FUNCTION_BLOCK "HF3_3#SB_FB2562"	// FB 2562
VERSION : 0.1
VAR_INPUT
  SCtrl : WORD ;	//上位控制命令
  inRD : ARRAY  [0 .. 3 ] OF //输入状态字
  WORD ;
  PT24 : TIME ;	//超时时间
  H_P_ALL_Ctrl : WORD ;	//全局控制命令
END_VAR
VAR_OUTPUT
  qnWR : WORD ;	//控制命令
  ToHMI1 : WORD ;	//反馈上位信息1
  ToHMI2 : WORD ;	//反馈上位信息2
  RT1 : INT ;	//1泵运行时间
  RT2 : INT ;	//2泵运行时间
  RT3 : INT ;
  SumFlt1 : INT ;	//1泵故障次数
  SumFlt2 : INT ;	//2泵故障次数
  SumFlt3 : INT ;
  SumRun1 : INT ;	//1泵运行次数
  SumRun2 : INT ;	//2泵运行次数
  SumRun3 : INT ;
  Level_Value : INT ;	//水位mm
END_VAR
VAR
  Ton1 : SFB 4;
  Ton2 : SFB 4;
  Ton3 : SFB 4;
  Ton4 : SFB 4;
  Ton5 : SFB 4;
  Ton6 : SFB 4;
  Ton7 : SFB 4;
  SingTout1 : BOOL ;	//一泵控制超时
  SingTout2 : BOOL ;	//二泵控制超时
  SingTout3 : BOOL ;	//三泵控制超时
  Timeout1 : BOOL ;	//一泵超时
  Timeout2 : BOOL ;	//二泵超时
  Timeout3 : BOOL ;	//三泵超时
  DI_Temp1 : ARRAY  [0 .. 15 ] OF //0自动1-1运行5-2运行9-3运行
  BOOL ;
  DI_Temp2 : ARRAY  [0 .. 15 ] OF //水泵状态字
  BOOL ;
  DO_Temp : ARRAY  [0 .. 15 ] OF //01-1泵启停23-2泵启停45-3泵启停
  BOOL ;
  Ctrl : ARRAY  [0 .. 15 ] OF //01-1泵启停23-2泵启停45-3泵启停
  BOOL ;
  SCtrl_Temp : ARRAY  [0 .. 15 ] OF //01-1泵启停23-2泵启停45-3泵启停6-3泵同启
  BOOL ;
  Latch : ARRAY  [0 .. 7 ] OF //01-1泵启停锁定23-2泵启停锁定45-3泵启停锁定
  BOOL ;
  McFlag : BOOL ;	//挂检修牌
  QTout1 : BOOL ;	//一泵输出超时
  QTout2 : BOOL ;	//二泵输出超时
  QTout3 : BOOL ;	//三泵输出超时
  H_P_ALL_Ctrl_Temp : ARRAY  [0 .. 15 ] OF BOOL ;
  CommOK_Temp : ARRAY  [0 .. 15 ] OF //通信中间变量
  BOOL ;
  CommOK : BOOL ;	//通信正常
END_VAR
BEGIN
NETWORK
TITLE =
      A(;
      BLD   1;
      =     L 4.0;
      TAR2  LD 0;
      L     #SCtrl;
      T     LW 5;
      L     DINO;
      T     LW 7;
      +AR2  P#206.0;
      TAR2;
      LAR2  LD 0;
      T     LD 9;
      UC    "HF3_W_T_B_FC54";
      {     P#L 5.0, P#L 7.0 };
      LAR2  LD 0;
      BLD   2;
      A     BR;
      );
      JNB   _001;
      BLD   1;
      =     L 4.0;
      TAR2  LD 0;
      L     #H_P_ALL_Ctrl;
      T     LW 5;
      L     DINO;
      T     LW 7;
      +AR2  P#212.0;
      TAR2;
      LAR2  LD 0;
      T     LD 9;
      UC    "HF3_W_T_B_FC54";
      {     P#L 5.0, P#L 7.0 };
      LAR2  LD 0;
      BLD   2;
_001: NOP   0;
NETWORK
TITLE =
      A(;
      BLD   1;
      =     L 4.0;
      TAR2  LD 0;
      L     #inRD[1];
      T     LW 5;
      L     DINO;
      T     LW 7;
      +AR2  P#198.0;
      TAR2;
      LAR2  LD 0;
      T     LD 9;
      UC    "HF3_W_T_B_FC54";
      {     P#L 5.0, P#L 7.0 };
      LAR2  LD 0;
      BLD   2;
      A     BR;
      );
      JNB   _002;
      BLD   1;
      =     L 4.0;
      TAR2  LD 0;
      L     #inRD[2];
      T     LW 5;
      L     DINO;
      T     LW 7;
      +AR2  P#200.0;
      TAR2;
      LAR2  LD 0;
      T     LD 9;
      UC    "HF3_W_T_B_FC54";
      {     P#L 5.0, P#L 7.0 };
      LAR2  LD 0;
      BLD   2;
_002: NOP   0;
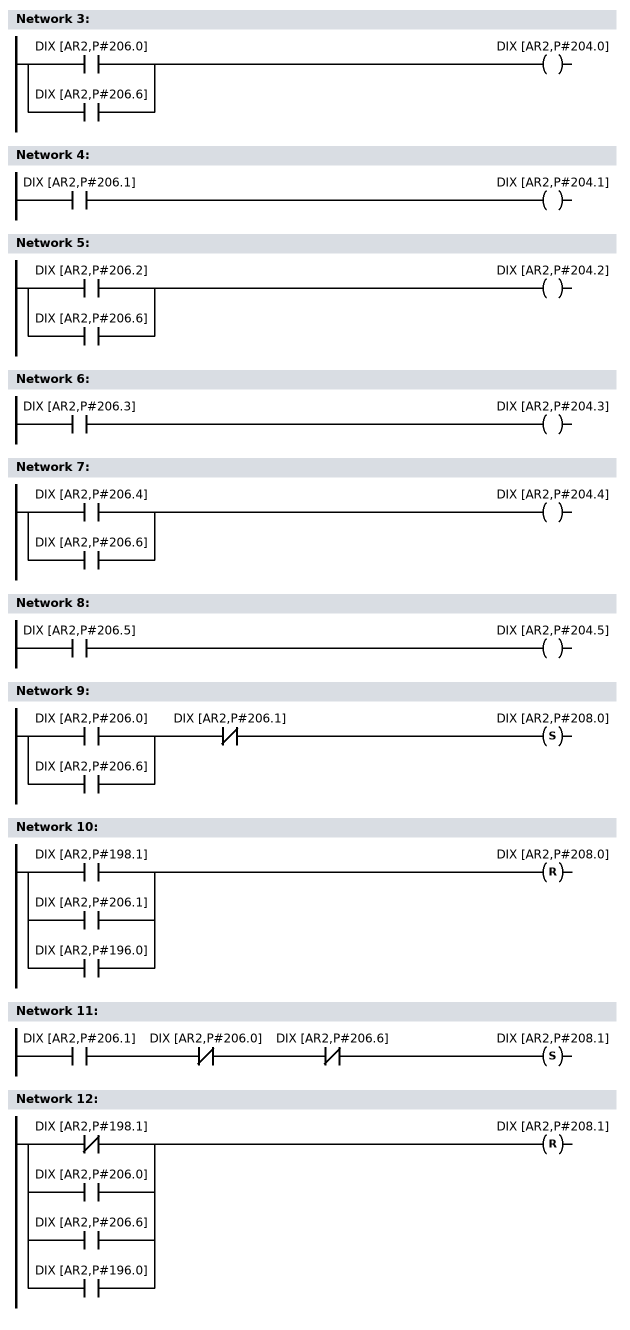
NETWORK
TITLE =
      O     DIX [AR2,P#206.0];
      O     DIX [AR2,P#206.6];
      =     DIX [AR2,P#204.0];
NETWORK
TITLE =
      A     DIX [AR2,P#206.1];
      =     DIX [AR2,P#204.1];
NETWORK
TITLE =
      O     DIX [AR2,P#206.2];
      O     DIX [AR2,P#206.6];
      =     DIX [AR2,P#204.2];
NETWORK
TITLE =
      A     DIX [AR2,P#206.3];
      =     DIX [AR2,P#204.3];
NETWORK
TITLE =
      O     DIX [AR2,P#206.4];
      O     DIX [AR2,P#206.6];
      =     DIX [AR2,P#204.4];
NETWORK
TITLE =
      A     DIX [AR2,P#206.5];
      =     DIX [AR2,P#204.5];
NETWORK
TITLE =
      A(;
      O     DIX [AR2,P#206.0];
      O     DIX [AR2,P#206.6];
      );
      AN    DIX [AR2,P#206.1];
      S     DIX [AR2,P#208.0];
NETWORK
TITLE =
      O     DIX [AR2,P#198.1];
      O     DIX [AR2,P#206.1];
      O     DIX [AR2,P#196.0];
      R     DIX [AR2,P#208.0];
NETWORK
TITLE =
      A     DIX [AR2,P#206.1];
      AN    DIX [AR2,P#206.0];
      AN    DIX [AR2,P#206.6];
      S     DIX [AR2,P#208.1];
NETWORK
TITLE =
      ON    DIX [AR2,P#198.1];
      O     DIX [AR2,P#206.0];
      O     DIX [AR2,P#206.6];
      O     DIX [AR2,P#196.0];
      R     DIX [AR2,P#208.1];
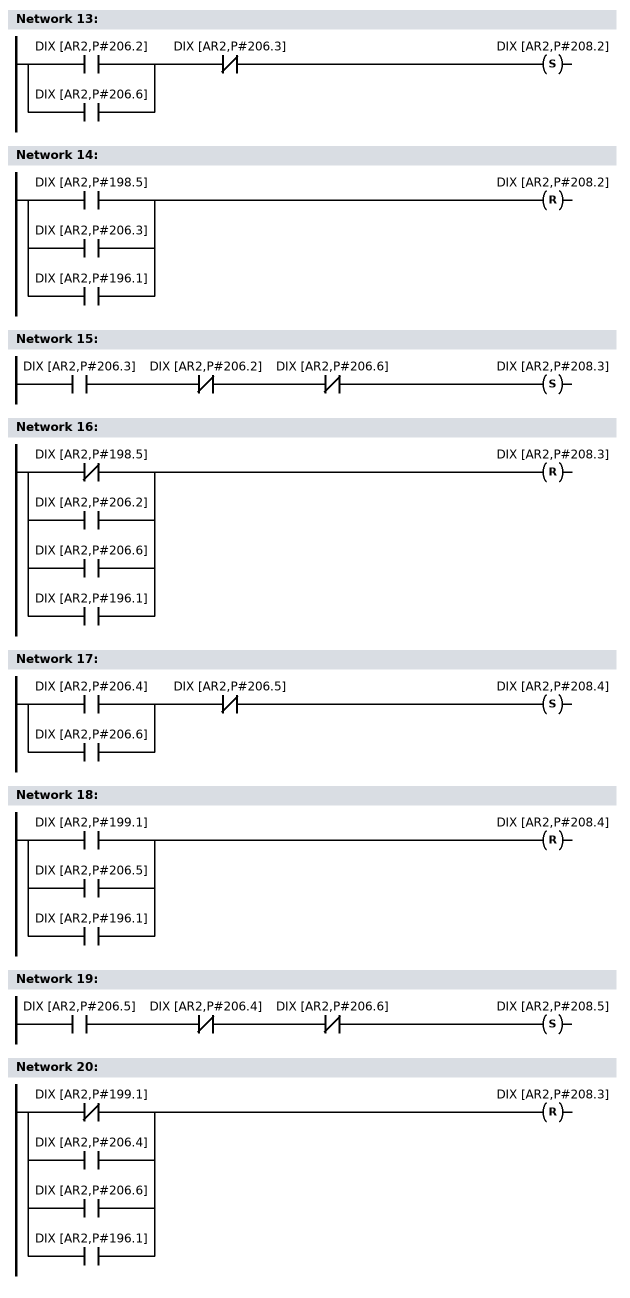
NETWORK
TITLE =
      A(;
      O     DIX [AR2,P#206.2];
      O     DIX [AR2,P#206.6];
      );
      AN    DIX [AR2,P#206.3];
      S     DIX [AR2,P#208.2];
NETWORK
TITLE =
      O     DIX [AR2,P#198.5];
      O     DIX [AR2,P#206.3];
      O     DIX [AR2,P#196.1];
      R     DIX [AR2,P#208.2];
NETWORK
TITLE =
      A     DIX [AR2,P#206.3];
      AN    DIX [AR2,P#206.2];
      AN    DIX [AR2,P#206.6];
      S     DIX [AR2,P#208.3];
NETWORK
TITLE =
      ON    DIX [AR2,P#198.5];
      O     DIX [AR2,P#206.2];
      O     DIX [AR2,P#206.6];
      O     DIX [AR2,P#196.1];
      R     DIX [AR2,P#208.3];
NETWORK
TITLE =
      A(;
      O     DIX [AR2,P#206.4];
      O     DIX [AR2,P#206.6];
      );
      AN    DIX [AR2,P#206.5];
      S     DIX [AR2,P#208.4];
NETWORK
TITLE =
      O     DIX [AR2,P#199.1];
      O     DIX [AR2,P#206.5];
      O     DIX [AR2,P#196.1];
      R     DIX [AR2,P#208.4];
NETWORK
TITLE =
      A     DIX [AR2,P#206.5];
      AN    DIX [AR2,P#206.4];
      AN    DIX [AR2,P#206.6];
      S     DIX [AR2,P#208.5];
NETWORK
TITLE =
      ON    DIX [AR2,P#199.1];
      O     DIX [AR2,P#206.4];
      O     DIX [AR2,P#206.6];
      O     DIX [AR2,P#196.1];
      R     DIX [AR2,P#208.3];
NETWORK
TITLE =
      A(;
      O     DIX [AR2,P#208.0];
      O     DIX [AR2,P#208.1];
      );
      AN    DIX [AR2,P#206.0];
      AN    DIX [AR2,P#206.1];
      AN    DIX [AR2,P#206.6];
      =     L 0.0;
      BLD   103;
      BLD   16;
      =     L 7.0;
      L     DINO;
      T     LW 5;
      CDB;
      OPN   DI [LW 5];
      TAR2  LD 1;
      A     L 0.0;
      =     DIX [AR2,P#42.0];
      L     DBD [AR2,P#10.0];
      T     DID [AR2,P#44.0];
      +AR2  P#42.0;
      UC    "TON";
      LAR2  LD 1;
      A     DIX [AR2,P#48.0];
      =     DBX [AR2,P#196.0];
      CDB;
      BLD   17;
      NOP   0;
NETWORK
TITLE =
      A(;
      O     DIX [AR2,P#202.0];
      O     DIX [AR2,P#202.1];
      );
      =     L 0.0;
      BLD   103;
      BLD   16;
      =     L 7.0;
      L     DINO;
      T     LW 5;
      CDB;
      OPN   DI [LW 5];
      TAR2  LD 1;
      A     L 0.0;
      =     DIX [AR2,P#64.0];
      L     DBD [AR2,P#10.0];
      T     DID [AR2,P#66.0];
      +AR2  P#64.0;
      UC    "TON";
      LAR2  LD 1;
      A     DIX [AR2,P#70.0];
      =     DBX [AR2,P#210.1];
      CDB;
      BLD   17;
      NOP   0;
NETWORK
TITLE =
      A(;
      O     DIX [AR2,P#208.2];
      O     DIX [AR2,P#208.3];
      );
      AN    DIX [AR2,P#206.2];
      AN    DIX [AR2,P#206.3];
      AN    DIX [AR2,P#206.6];
      =     L 0.0;
      BLD   103;
      BLD   16;
      =     L 7.0;
      L     DINO;
      T     LW 5;
      CDB;
      OPN   DI [LW 5];
      TAR2  LD 1;
      A     L 0.0;
      =     DIX [AR2,P#86.0];
      L     DBD [AR2,P#10.0];
      T     DID [AR2,P#88.0];
      +AR2  P#86.0;
      UC    "TON";
      LAR2  LD 1;
      A     DIX [AR2,P#92.0];
      =     DBX [AR2,P#196.1];
      CDB;
      BLD   17;
      NOP   0;
NETWORK
TITLE =
      A(;
      O     DIX [AR2,P#202.2];
      O     DIX [AR2,P#202.3];
      );
      =     L 0.0;
      BLD   103;
      BLD   16;
      =     L 7.0;
      L     DINO;
      T     LW 5;
      CDB;
      OPN   DI [LW 5];
      TAR2  LD 1;
      A     L 0.0;
      =     DIX [AR2,P#108.0];
      L     DBD [AR2,P#10.0];
      T     DID [AR2,P#110.0];
      +AR2  P#108.0;
      UC    "TON";
      LAR2  LD 1;
      A     DIX [AR2,P#114.0];
      =     DBX [AR2,P#210.2];
      CDB;
      BLD   17;
      NOP   0;
NETWORK
TITLE =
      A(;
      O     DIX [AR2,P#208.4];
      O     DIX [AR2,P#208.5];
      );
      AN    DIX [AR2,P#206.4];
      AN    DIX [AR2,P#206.5];
      AN    DIX [AR2,P#206.6];
      =     L 0.0;
      BLD   103;
      BLD   16;
      =     L 7.0;
      L     DINO;
      T     LW 5;
      CDB;
      OPN   DI [LW 5];
      TAR2  LD 1;
      A     L 0.0;
      =     DIX [AR2,P#130.0];
      L     DBD [AR2,P#10.0];
      T     DID [AR2,P#132.0];
      +AR2  P#130.0;
      UC    "TON";
      LAR2  LD 1;
      A     DIX [AR2,P#136.0];
      =     DBX [AR2,P#196.2];
      CDB;
      BLD   17;
      NOP   0;
NETWORK
TITLE =
      A(;
      O     DIX [AR2,P#202.4];
      O     DIX [AR2,P#202.5];
      );
      =     L 0.0;
      BLD   103;
      BLD   16;
      =     L 7.0;
      L     DINO;
      T     LW 5;
      CDB;
      OPN   DI [LW 5];
      TAR2  LD 1;
      A     L 0.0;
      =     DIX [AR2,P#174.0];
      L     DBD [AR2,P#10.0];
      T     DID [AR2,P#176.0];
      +AR2  P#174.0;
      UC    "TON";
      LAR2  LD 1;
      A     DIX [AR2,P#180.0];
      =     DBX [AR2,P#210.3];
      CDB;
      BLD   17;
      NOP   0;
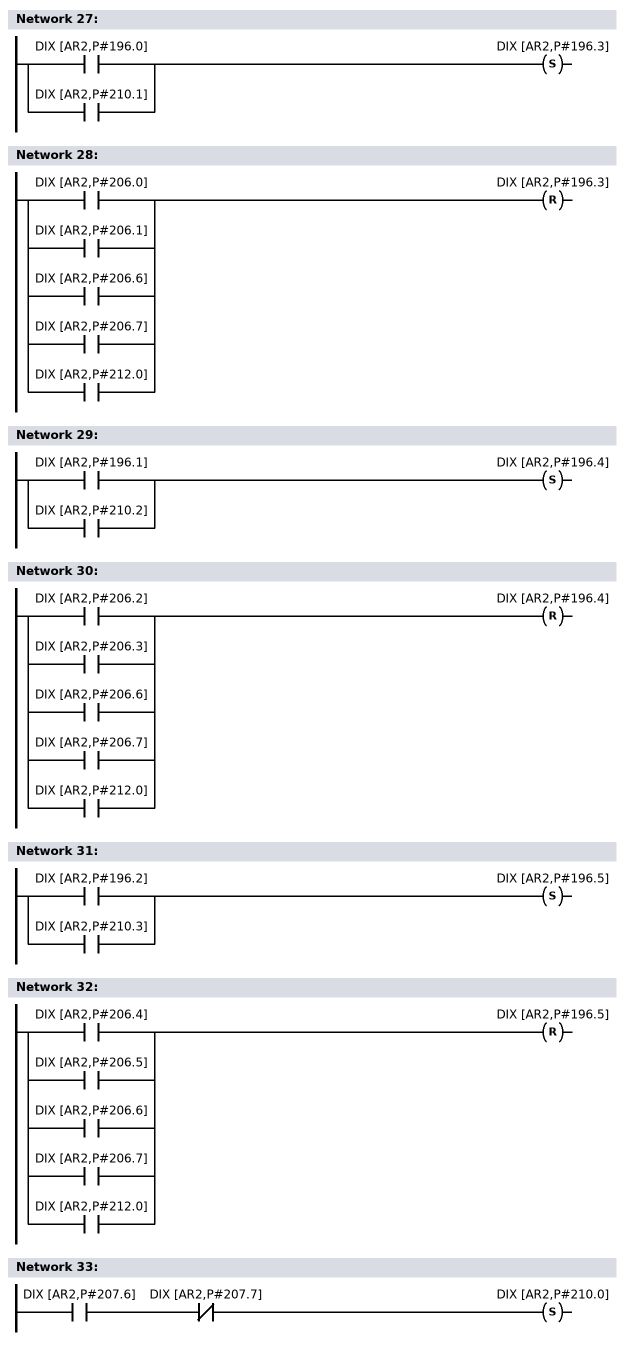
NETWORK
TITLE =
      O     DIX [AR2,P#196.0];
      O     DIX [AR2,P#210.1];
      S     DIX [AR2,P#196.3];
NETWORK
TITLE =
      O     DIX [AR2,P#206.0];
      O     DIX [AR2,P#206.1];
      O     DIX [AR2,P#206.6];
      O     DIX [AR2,P#206.7];
      O     DIX [AR2,P#212.0];
      R     DIX [AR2,P#196.3];
NETWORK
TITLE =
      O     DIX [AR2,P#196.1];
      O     DIX [AR2,P#210.2];
      S     DIX [AR2,P#196.4];
NETWORK
TITLE =
      O     DIX [AR2,P#206.2];
      O     DIX [AR2,P#206.3];
      O     DIX [AR2,P#206.6];
      O     DIX [AR2,P#206.7];
      O     DIX [AR2,P#212.0];
      R     DIX [AR2,P#196.4];
NETWORK
TITLE =
      O     DIX [AR2,P#196.2];
      O     DIX [AR2,P#210.3];
      S     DIX [AR2,P#196.5];
NETWORK
TITLE =
      O     DIX [AR2,P#206.4];
      O     DIX [AR2,P#206.5];
      O     DIX [AR2,P#206.6];
      O     DIX [AR2,P#206.7];
      O     DIX [AR2,P#212.0];
      R     DIX [AR2,P#196.5];
NETWORK
TITLE =
      A     DIX [AR2,P#207.6];
      AN    DIX [AR2,P#207.7];
      S     DIX [AR2,P#210.0];
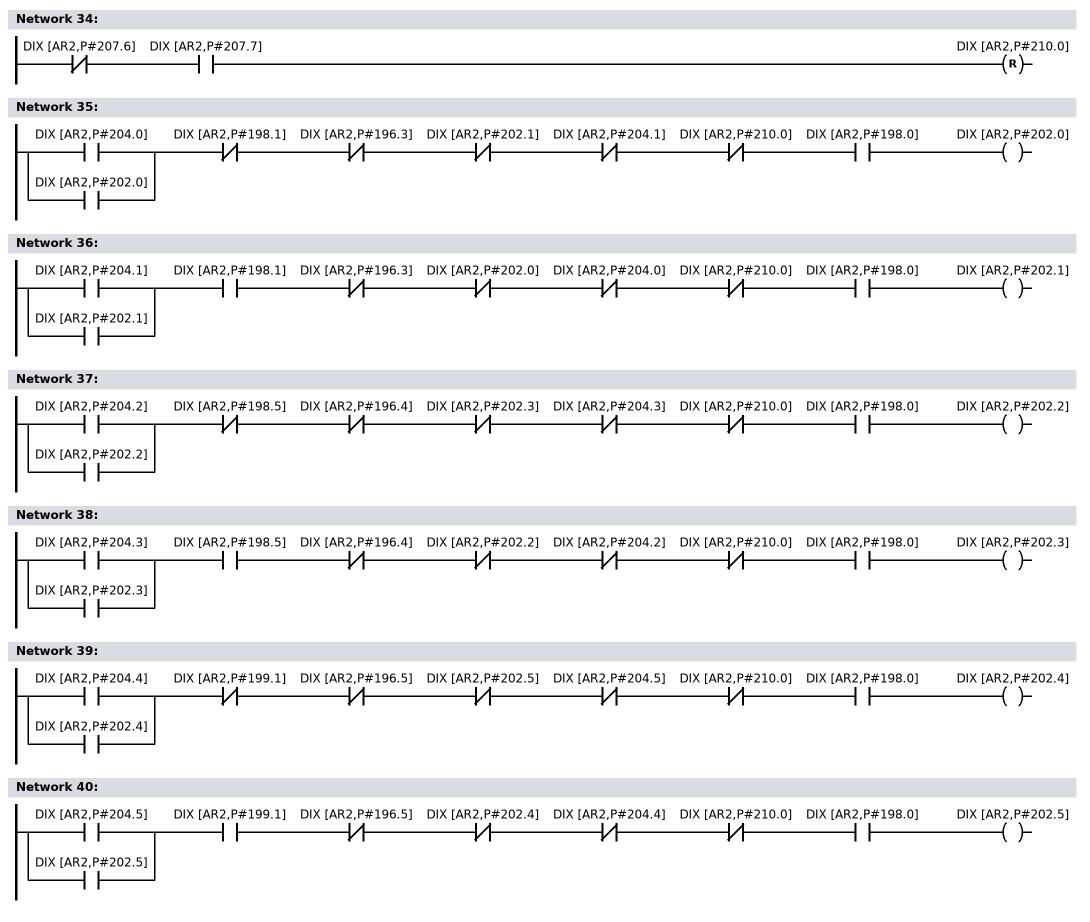
NETWORK
TITLE =
      AN    DIX [AR2,P#207.6];
      A     DIX [AR2,P#207.7];
      R     DIX [AR2,P#210.0];
NETWORK
TITLE =
      A(;
      O     DIX [AR2,P#204.0];
      O     DIX [AR2,P#202.0];
      );
      AN    DIX [AR2,P#198.1];
      AN    DIX [AR2,P#196.3];
      AN    DIX [AR2,P#202.1];
      AN    DIX [AR2,P#204.1];
      AN    DIX [AR2,P#210.0];
      A     DIX [AR2,P#198.0];
      =     DIX [AR2,P#202.0];
NETWORK
TITLE =
      A(;
      O     DIX [AR2,P#204.1];
      O     DIX [AR2,P#202.1];
      );
      A     DIX [AR2,P#198.1];
      AN    DIX [AR2,P#196.3];
      AN    DIX [AR2,P#202.0];
      AN    DIX [AR2,P#204.0];
      AN    DIX [AR2,P#210.0];
      A     DIX [AR2,P#198.0];
      =     DIX [AR2,P#202.1];
NETWORK
TITLE =
      A(;
      O     DIX [AR2,P#204.2];
      O     DIX [AR2,P#202.2];
      );
      AN    DIX [AR2,P#198.5];
      AN    DIX [AR2,P#196.4];
      AN    DIX [AR2,P#202.3];
      AN    DIX [AR2,P#204.3];
      AN    DIX [AR2,P#210.0];
      A     DIX [AR2,P#198.0];
      =     DIX [AR2,P#202.2];
NETWORK
TITLE =
      A(;
      O     DIX [AR2,P#204.3];
      O     DIX [AR2,P#202.3];
      );
      A     DIX [AR2,P#198.5];
      AN    DIX [AR2,P#196.4];
      AN    DIX [AR2,P#202.2];
      AN    DIX [AR2,P#204.2];
      AN    DIX [AR2,P#210.0];
      A     DIX [AR2,P#198.0];
      =     DIX [AR2,P#202.3];
NETWORK
TITLE =
      A(;
      O     DIX [AR2,P#204.4];
      O     DIX [AR2,P#202.4];
      );
      AN    DIX [AR2,P#199.1];
      AN    DIX [AR2,P#196.5];
      AN    DIX [AR2,P#202.5];
      AN    DIX [AR2,P#204.5];
      AN    DIX [AR2,P#210.0];
      A     DIX [AR2,P#198.0];
      =     DIX [AR2,P#202.4];
NETWORK
TITLE =
      A(;
      O     DIX [AR2,P#204.5];
      O     DIX [AR2,P#202.5];
      );
      A     DIX [AR2,P#199.1];
      AN    DIX [AR2,P#196.5];
      AN    DIX [AR2,P#202.4];
      AN    DIX [AR2,P#204.4];
      AN    DIX [AR2,P#210.0];
      A     DIX [AR2,P#198.0];
      =     DIX [AR2,P#202.5];
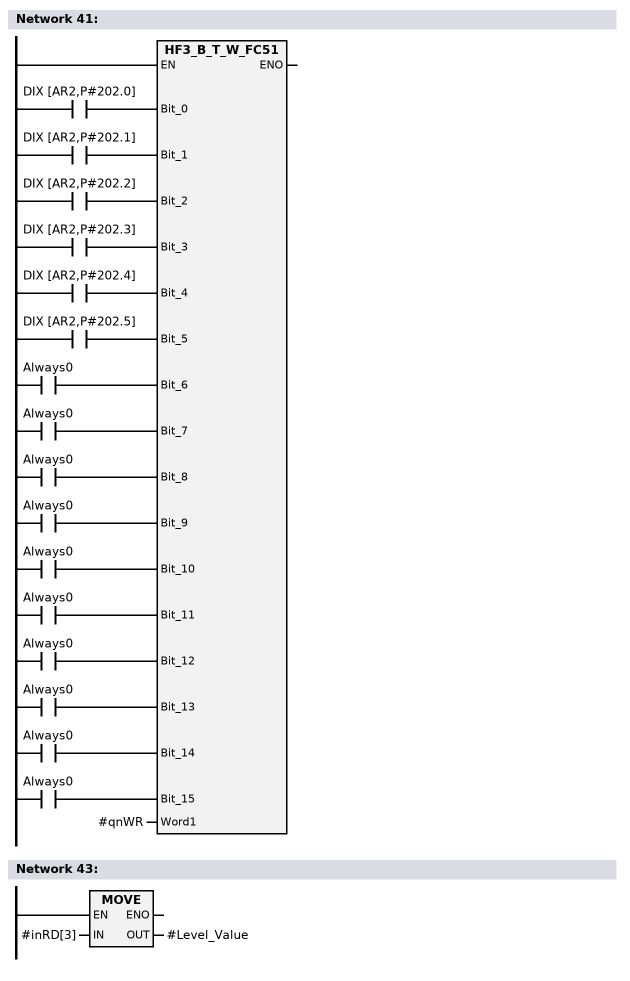
NETWORK
TITLE =
      A     DIX [AR2,P#202.0];
      =     L 0.0;
      BLD   103;
      A     DIX [AR2,P#202.1];
      =     L 0.1;
      BLD   103;
      A     DIX [AR2,P#202.2];
      =     L 0.2;
      BLD   103;
      A     DIX [AR2,P#202.3];
      =     L 0.3;
      BLD   103;
      A     DIX [AR2,P#202.4];
      =     L 0.4;
      BLD   103;
      A     DIX [AR2,P#202.5];
      =     L 0.5;
      BLD   103;
      A     "Always0";
      =     L 0.6;
      BLD   103;
      A     "Always0";
      =     L 0.7;
      BLD   103;
      A     "Always0";
      =     L 1.0;
      BLD   103;
      A     "Always0";
      =     L 1.1;
      BLD   103;
      A     "Always0";
      =     L 1.2;
      BLD   103;
      A     "Always0";
      =     L 1.3;
      BLD   103;
      A     "Always0";
      =     L 1.4;
      BLD   103;
      A     "Always0";
      =     L 1.5;
      BLD   103;
      A     "Always0";
      =     L 1.6;
      BLD   103;
      A     "Always0";
      =     L 1.7;
      BLD   103;
      CALL  "HF3_B_T_W_FC51" (
           Bit_0                    := L 0.0,
           Bit_1                    := L 0.1,
           Bit_2                    := L 0.2,
           Bit_3                    := L 0.3,
           Bit_4                    := L 0.4,
           Bit_5                    := L 0.5,
           Bit_6                    := L 0.6,
           Bit_7                    := L 0.7,
           Bit_8                    := L 1.0,
           Bit_9                    := L 1.1,
           Bit_10                   := L 1.2,
           Bit_11                   := L 1.3,
           Bit_12                   := L 1.4,
           Bit_13                   := L 1.5,
           Bit_14                   := L 1.6,
           Bit_15                   := L 1.7,
           Word1                    := #qnWR);
      NOP   0;
NETWORK
TITLE =
      A     "Always0";
      =     L 0.0;
      BLD   103;
      A     DIX [AR2,P#198.5];
      =     L 0.1;
      BLD   103;
      A     DIX [AR2,P#198.6];
      =     L 0.2;
      BLD   103;
      A     DIX [AR2,P#198.7];
      =     L 0.3;
      BLD   103;
      A     DIX [AR2,P#199.0];
      =     L 0.4;
      BLD   103;
      A     DIX [AR2,P#199.1];
      =     L 0.5;
      BLD   103;
      A     DIX [AR2,P#199.2];
      =     L 0.6;
      BLD   103;
      A     DIX [AR2,P#199.3];
      =     L 0.7;
      BLD   103;
      A     DIX [AR2,P#199.4];
      =     L 1.0;
      BLD   103;
      A     DIX [AR2,P#199.7];
      =     L 1.1;
      BLD   103;
      A     DIX [AR2,P#199.6];
      =     L 1.2;
      BLD   103;
      A     "Always0";
      =     L 1.3;
      BLD   103;
      A     "Always0";
      =     L 1.4;
      BLD   103;
      A     "Always0";
      =     L 1.5;
      BLD   103;
      A     "Always0";
      =     L 1.6;
      BLD   103;
      A     "Always0";
      =     L 1.7;
      BLD   103;
      A(;
      A     DIX [AR2,P#198.0];
      =     L 2.0;
      BLD   103;
      A     DIX [AR2,P#198.1];
      =     L 2.1;
      BLD   103;
      A     DIX [AR2,P#198.2];
      =     L 2.2;
      BLD   103;
      A     DIX [AR2,P#198.3];
      =     L 2.3;
      BLD   103;
      A     DIX [AR2,P#198.4];
      =     L 2.4;
      BLD   103;
      A     DIX [AR2,P#200.0];
      =     L 2.5;
      BLD   103;
      A     DIX [AR2,P#199.5];
      =     L 2.6;
      BLD   103;
      A     DIX [AR2,P#200.1];
      =     L 2.7;
      BLD   103;
      A     DIX [AR2,P#200.2];
      =     L 3.0;
      BLD   103;
      A     "Always0";
      =     L 3.1;
      BLD   103;
      A     "Always0";
      =     L 3.2;
      BLD   103;
      A     DIX [AR2,P#196.3];
      =     L 3.3;
      BLD   103;
      A     DIX [AR2,P#196.4];
      =     L 3.4;
      BLD   103;
      A     DIX [AR2,P#196.5];
      =     L 3.5;
      BLD   103;
      A     DIX [AR2,P#210.0];
      =     L 3.6;
      BLD   103;
      A     DIX [AR2,P#216.0];
      =     L 3.7;
      BLD   103;
      CALL  "HF3_B_T_W_FC51" (
           Bit_0                    := L 2.0,
           Bit_1                    := L 2.1,
           Bit_2                    := L 2.2,
           Bit_3                    := L 2.3,
           Bit_4                    := L 2.4,
           Bit_5                    := L 2.5,
           Bit_6                    := L 2.6,
           Bit_7                    := L 2.7,
           Bit_8                    := L 3.0,
           Bit_9                    := L 3.1,
           Bit_10                   := L 3.2,
           Bit_11                   := L 3.3,
           Bit_12                   := L 3.4,
           Bit_13                   := L 3.5,
           Bit_14                   := L 3.6,
           Bit_15                   := L 3.7,
           Word1                    := #ToHMI1);
      A     BR;
      );
      JNB   _003;
      CALL  "HF3_B_T_W_FC51" (
           Bit_0                    := L 0.0,
           Bit_1                    := L 0.1,
           Bit_2                    := L 0.2,
           Bit_3                    := L 0.3,
           Bit_4                    := L 0.4,
           Bit_5                    := L 0.5,
           Bit_6                    := L 0.6,
           Bit_7                    := L 0.7,
           Bit_8                    := L 1.0,
           Bit_9                    := L 1.1,
           Bit_10                   := L 1.2,
           Bit_11                   := L 1.3,
           Bit_12                   := L 1.4,
           Bit_13                   := L 1.5,
           Bit_14                   := L 1.6,
           Bit_15                   := L 1.7,
           Word1                    := #ToHMI2);
_003: NOP   0;
NETWORK
TITLE =
      L     #inRD[3];
      T     #Level_Value;
      NOP   0;
NETWORK
TITLE =
      BLD   1;
      =     L 4.0;
      TAR2  LD 0;
      L     #inRD[0];
      T     LW 5;
      L     DINO;
      T     LW 7;
      +AR2  P#214.0;
      TAR2;
      LAR2  LD 0;
      T     LD 9;
      UC    "HF3_W_T_B_FC54";
      {     P#L 5.0, P#L 7.0 };
      LAR2  LD 0;
      BLD   2;
      NOP   0;
NETWORK
TITLE =
      A(;
      O     DIX [AR2,P#214.0];
      ON    DIX [AR2,P#214.0];
      );
      =     L 0.0;
      BLD   103;
      BLD   16;
      =     L 7.0;
      L     DINO;
      T     LW 5;
      CDB;
      OPN   DI [LW 5];
      TAR2  LD 1;
      A     L 0.0;
      =     DIX [AR2,P#130.0];
      L     L#3000;
      T     DID [AR2,P#132.0];
      +AR2  P#130.0;
      UC    "TON";
      LAR2  LD 1;
      A     DIX [AR2,P#136.0];
      =     DBX [AR2,P#216.0];
      CDB;
      BLD   17;
      NOP   0;
END_FUNCTION_BLOCK

FUNCTION_BLOCK "HF3_WSB_FB2581"	// FB 2581
VERSION : 0.1
VAR
  AP_03 : FB 2582;
END_VAR
BEGIN
NETWORK
TITLE =
      BLD   14;
      =     L 6.0;
      L     DINO;
      T     LW 4;
      CDB;
      OPN   DI [LW 4];
      TAR2  LD 0;
      OPN   DI 2265;
      L     DIW 2;
      OPN   DI [LW 4];
      T     #AP_03.DB_NO;
      OPN   DI 2265;
      L     DIW 6;
      OPN   DI [LW 4];
      T     DIW [AR2,P#2.0];
      +AR2  P#0.0;
      UC    "HF3_WSB_FB2582";
      LAR2  LD 0;
      L     #AP_03.in_stradr;
      OPN   DI 6002;
      T     DIW 336;
      OPN   DI [LW 4];
      L     #AP_03.Level_Value;
      OPN   DI 6002;
      T     DIW 338;
      OPN   DI [LW 4];
      CDB;
      BLD   15;
      NOP   0;
END_FUNCTION_BLOCK

FUNCTION_BLOCK "HF3_WSB_FB2582"	// FB 2582
VERSION : 0.1
VAR_INPUT
  DB_NO : INT ;	//读DB号
  Multi : BOOL ;	//是否有多个水泵并线
  in_stradr : INT ;	//读命令状态开始地址
END_VAR
VAR_OUTPUT
  Level_Value : INT ;
  ToHMI : WORD ;
END_VAR
VAR
  IN_RD1 : WORD ;
  IN_RD2 : WORD ;
  COMM_HB : WORD ;
  DI_Temp1 : ARRAY  [0 .. 15 ] OF BOOL ;
  DI_Temp2 : ARRAY  [0 .. 15 ] OF BOOL ;
  CommOK_Temp : BOOL ;
  CommOK : BOOL ;
  Ton1 : SFB 4;
END_VAR
VAR_TEMP
  DI_reg : INT ;
  db_no_temp : INT ;
  AR2_VALUE : DWORD ;	//AR2寄存器原始值
END_VAR
BEGIN
NETWORK
TITLE =
      CLR;
      L     #DB_NO;
      T     #db_no_temp;
//当CP340接入多个水泵时
      L     P#0.0;
      LAR1;
      A     #Multi;
      JCN   sigl;
      L     #in_stradr;
      SLD   3;
      LAR1;
// AR1用于访问DB AR2用于访问DIB
//sigl: TAR2  
//    T     #AR2_VALUE
//   AD    DW#16#FFFFFF
//  L     P##IN_RD1
//   +D    
//  LAR2  
// 寄存器40204 、40205内容传递 通讯状态传递
sigl: OPN   DB [#db_no_temp];	//寄存器40204内容传递
      L     DBW [AR1,P#8.0];
// T     W [AR2,P#0.0]
      T     #IN_RD1;
      L     DBW [AR1,P#10.0];	//寄存器40205内容传递
// T     W [AR2,P#2.0]
      T     #IN_RD2;
      L     DBW [AR1,P#0.0];
//  T     W [AR2,P#4.0]               //该设备通讯状态   0为正常
      T     #COMM_HB;
//水泵水位数值传递
//    L     #AR2_VALUE
//  AD    DW#16#FFFFFF
//    L     P##Level_Value
//   +D    
//  LAR2                              //寄存器40201
      L     DBW [AR1,P#2.0];
//  T     W [AR2,P#0.0]               // 水泵水位赋值
      T     #Level_Value;
//恢复AR2中的初始值
//     L     #AR2_VALUE
//    LAR2  
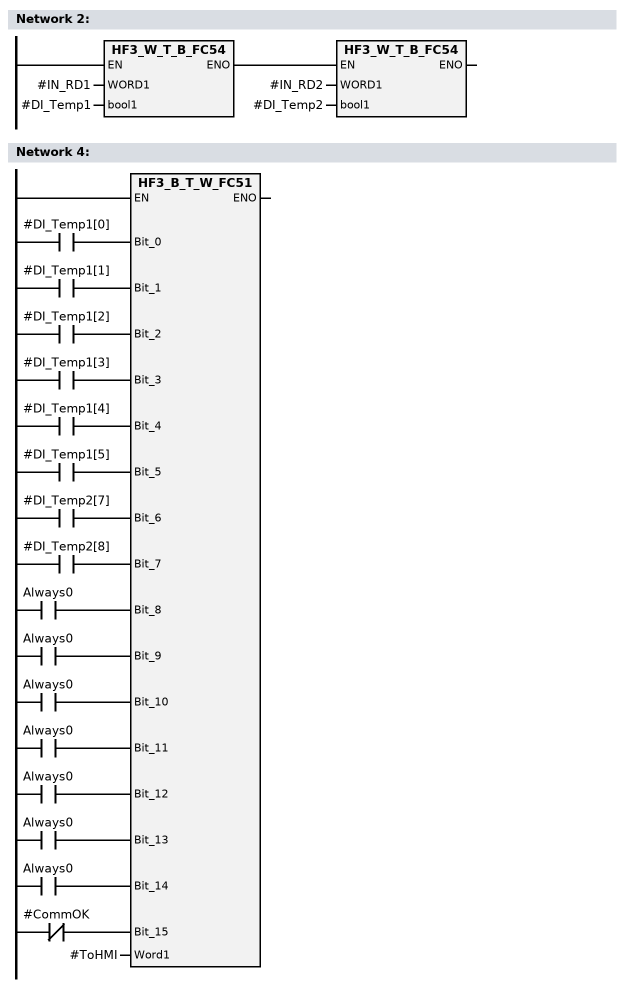
NETWORK
TITLE =
      A(;
      CALL  "HF3_W_T_B_FC54" (
           WORD1                    := #IN_RD1,
           bool1                    := #DI_Temp1);
      A     BR;
      );
      JNB   _001;
      CALL  "HF3_W_T_B_FC54" (
           WORD1                    := #IN_RD2,
           bool1                    := #DI_Temp2);
_001: NOP   0;
NETWORK
TITLE =
      CLR;
      L     #COMM_HB;
      L     W#16#0;
      <>I;
      =     #CommOK_Temp;
      BLD   16;
      =     L 14.0;
      L     DINO;
      T     LW 12;
      CDB;
      OPN   DI [LW 12];
      TAR2  LD 8;
      A     DBX [AR2,P#20.0];
      =     DIX [AR2,P#22.0];
      L     L#3000;
      T     DID [AR2,P#24.0];
      +AR2  P#22.0;
      UC    "TON";
      LAR2  LD 8;
      A     DIX [AR2,P#28.0];
      =     DBX [AR2,P#20.1];
      CDB;
      BLD   17;
NETWORK
TITLE =
      A     #DI_Temp1[0];
      =     L 8.0;
      BLD   103;
      A     #DI_Temp1[1];
      =     L 8.1;
      BLD   103;
      A     #DI_Temp1[2];
      =     L 8.2;
      BLD   103;
      A     #DI_Temp1[3];
      =     L 8.3;
      BLD   103;
      A     #DI_Temp1[4];
      =     L 8.4;
      BLD   103;
      A     #DI_Temp1[5];
      =     L 8.5;
      BLD   103;
      A     #DI_Temp2[7];
      =     L 8.6;
      BLD   103;
      A     #DI_Temp2[8];
      =     L 8.7;
      BLD   103;
      A     "Always0";
      =     L 9.0;
      BLD   103;
      A     "Always0";
      =     L 9.1;
      BLD   103;
      A     "Always0";
      =     L 9.2;
      BLD   103;
      A     "Always0";
      =     L 9.3;
      BLD   103;
      A     "Always0";
      =     L 9.4;
      BLD   103;
      A     "Always0";
      =     L 9.5;
      BLD   103;
      A     "Always0";
      =     L 9.6;
      BLD   103;
      AN    #CommOK;
      =     L 9.7;
      BLD   103;
      CALL  "HF3_B_T_W_FC51" (
           Bit_0                    := L 8.0,
           Bit_1                    := L 8.1,
           Bit_2                    := L 8.2,
           Bit_3                    := L 8.3,
           Bit_4                    := L 8.4,
           Bit_5                    := L 8.5,
           Bit_6                    := L 8.6,
           Bit_7                    := L 8.7,
           Bit_8                    := L 9.0,
           Bit_9                    := L 9.1,
           Bit_10                   := L 9.2,
           Bit_11                   := L 9.3,
           Bit_12                   := L 9.4,
           Bit_13                   := L 9.5,
           Bit_14                   := L 9.6,
           Bit_15                   := L 9.7,
           Word1                    := #ToHMI);
      NOP   0;
END_FUNCTION_BLOCK

FUNCTION_BLOCK "HF3_PSB_FB2591"	// FB 2591
VERSION : 0.1
VAR
  AP_PSB_B : FB 2592;
  AP_PSB_C : FB 2592;
  AP_FSB_1 : FB 2592;
  AP_PSB_2 : FB 2592;
END_VAR
BEGIN
NETWORK
TITLE = AP_PSB_B
      A     "Always0";
      =     L 0.0;
      BLD   103;
      BLD   14;
      =     L 7.0;
      L     DINO;
      T     LW 5;
      CDB;
      OPN   DI [LW 5];
      TAR2  LD 1;
      L     2;
      T     #AP_PSB_B.number;
      L     2005;
      T     #AP_PSB_B.DB_NO;
      A     L 0.0;
      =     #AP_PSB_B.Multi;
      L     0;
      T     #AP_PSB_B.in_stradr;
      +AR2  P#0.0;
      UC    "HF3_PSB_FB2592";
      LAR2  LD 1;
      L     #AP_PSB_B.Level_Value;
      OPN   DI 6004;
      T     DIW 24;
      OPN   DI [LW 5];
      L     #AP_PSB_B.ToHMI;
      OPN   DI 6004;
      T     DIW 22;
      OPN   DI [LW 5];
      CDB;
      BLD   15;
      NOP   0;
NETWORK
TITLE = AP_PSB_C
      A     "Always0";
      =     L 0.0;
      BLD   103;
      BLD   14;
      =     L 7.0;
      L     DINO;
      T     LW 5;
      CDB;
      OPN   DI [LW 5];
      TAR2  LD 1;
      L     2;
      T     DIW [AR2,P#46.0];
      L     2075;
      T     DIW [AR2,P#48.0];
      A     L 0.0;
      =     DIX [AR2,P#50.0];
      L     0;
      T     DIW [AR2,P#52.0];
      +AR2  P#46.0;
      UC    "HF3_PSB_FB2592";
      LAR2  LD 1;
      L     DIW [AR2,P#54.0];
      OPN   DI 6004;
      T     DIW 28;
      OPN   DI [LW 5];
      L     DIW [AR2,P#56.0];
      OPN   DI 6004;
      T     DIW 26;
      OPN   DI [LW 5];
      CDB;
      BLD   15;
      NOP   0;
NETWORK
TITLE = AP_FSB1
      A     "Always1";
      =     L 0.0;
      BLD   103;
      BLD   14;
      =     L 7.0;
      L     DINO;
      T     LW 5;
      CDB;
      OPN   DI [LW 5];
      TAR2  LD 1;
      L     2;
      T     DIW [AR2,P#92.0];
      L     2065;
      T     DIW [AR2,P#94.0];
      A     L 0.0;
      =     DIX [AR2,P#96.0];
      L     24;
      T     DIW [AR2,P#98.0];
      +AR2  P#92.0;
      UC    "HF3_PSB_FB2592";
      LAR2  LD 1;
      L     DIW [AR2,P#100.0];
      OPN   DI 6004;
      T     DIW 32;
      OPN   DI [LW 5];
      L     DIW [AR2,P#102.0];
      OPN   DI 6004;
      T     DIW 30;
      OPN   DI [LW 5];
      CDB;
      BLD   15;
      NOP   0;
NETWORK
TITLE = AP_FSB2
NETWORK
TITLE =
END_FUNCTION_BLOCK

FUNCTION_BLOCK "HF3_PSB_FB2592"	// FB 2592
TITLE = 局部排水泵
//不要修改STL程序 不要改变IN OUT STAT 引脚参数在接口里的顺序
VERSION : 0.1
VAR_INPUT
  number : INT ;	//单泵填1，双泵填2
  DB_NO : INT ;	//读DB号
  Multi : BOOL ;	//是否有多个水泵并线
  in_stradr : INT ;	//读命令状态开始地址
END_VAR
VAR_OUTPUT
  Level_Value : INT ;
  ToHMI : WORD ;
END_VAR
VAR
  TON1 : SFB 4;
  IN_RD1 : WORD ;
  IN_RD2 : WORD ;
  Comm_HB : WORD ;
  DI_Temp1 : ARRAY  [0 .. 15 ] OF BOOL ;
  DI_Temp2 : ARRAY  [0 .. 15 ] OF BOOL ;
  CommOK_Temp : BOOL ;
  CommOK : BOOL ;
END_VAR
VAR_TEMP
  DI_reg : INT ;
  db_no_temp : INT ;
  AR2_VALUE : DWORD ;	//AR2寄存器原始值
END_VAR
BEGIN
NETWORK
TITLE = 状态信息读取
      CLR;
      L     #DB_NO;
      T     #db_no_temp;
//当CP340接入多个水泵时
      L     P#0.0;
      LAR1;
      A     #Multi;
      JCN   sigl;
      L     #in_stradr;
      SLD   3;
      LAR1;
// AR1用于访问DB AR2用于访问DIB
//sigl: TAR2  
//    T     #AR2_VALUE
//    AD    DW#16#FFFFFF
//   L     P##IN_RD1
//   +D    
//  LAR2  
// 寄存器40002 、40003内容传递 通讯状态传递
sigl: OPN   DB [#db_no_temp];	//寄存器40002内容传递
      L     DBW [AR1,P#4.0];
//    T     W [AR2,P#0.0]
      T     DIW [AR2,P#34.0];
      L     DBW [AR1,P#6.0];	//寄存器40003内容传递
//     T     W [AR2,P#2.0]
      T     DIW [AR2,P#36.0];
      L     DBW [AR1,P#0.0];
//   T     W [AR2,P#4.0]               //该设备通讯状态   0为正常
      T     DIW [AR2,P#38.0];
//水泵水位数值传递
//    L     #AR2_VALUE
//   AD    DW#16#FFFFFF
//   L     P##Level_Value
//    +D    
//   LAR2  
      L     DBW [AR1,P#8.0];
// T     W [AR2,P#0.0]               // 水泵水位赋值
      T     #Level_Value;
//恢复AR2中的初始值
//     L     #AR2_VALUE
//    LAR2  
NETWORK
TITLE = 寄存器信息分解
      A(;
      BLD   1;
      =     L 12.0;
      TAR2  LD 8;
      L     DIW [AR2,P#34.0];
      T     LW 13;
      L     DINO;
      T     LW 15;
      +AR2  P#40.0;
      TAR2;
      LAR2  LD 8;
      T     LD 17;
      UC    "HF3_W_T_B_FC54";
      {     P#L 13.0, P#L 15.0 };
      LAR2  LD 8;
      BLD   2;
      A     BR;
      );
      JNB   _001;
      BLD   1;
      =     L 12.0;
      TAR2  LD 8;
      L     DIW [AR2,P#36.0];
      T     LW 13;
      L     DINO;
      T     LW 15;
      +AR2  P#42.0;
      TAR2;
      LAR2  LD 8;
      T     LD 17;
      UC    "HF3_W_T_B_FC54";
      {     P#L 13.0, P#L 15.0 };
      LAR2  LD 8;
      BLD   2;
_001: NOP   0;
NETWORK
TITLE = 通讯状态判断
      CLR;
      L     DIW [AR2,P#38.0];
      L     W#16#0;
      <>I;
      =     DIX [AR2,P#44.0];
      BLD   16;
      =     L 14.0;
      L     DINO;
      T     LW 12;
      CDB;
      OPN   DI [LW 12];
      TAR2  LD 8;
      A     DBX [AR2,P#44.0];
      =     DIX [AR2,P#12.0];
      L     L#3000;
      T     DID [AR2,P#14.0];
      +AR2  P#12.0;
      UC    "TON";
      LAR2  LD 8;
      A     DIX [AR2,P#18.0];
      =     DBX [AR2,P#44.1];
      CDB;
      BLD   17;
NETWORK
TITLE = 水泵单双泵类型
      CLR;
      L     #number;
      L     W#16#2;
      ==I;
// 双泵时跳转
      JC    PUM2;
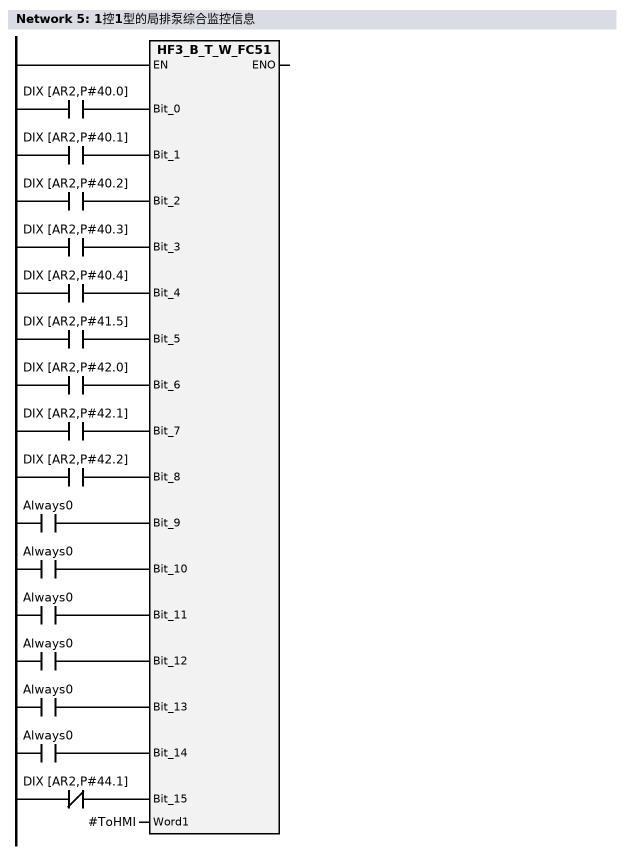
NETWORK
TITLE = 1控1型的局排泵综合监控信息
      A     DIX [AR2,P#40.0];
      =     L 8.0;
      BLD   103;
      A     DIX [AR2,P#40.1];
      =     L 8.1;
      BLD   103;
      A     DIX [AR2,P#40.2];
      =     L 8.2;
      BLD   103;
      A     DIX [AR2,P#40.3];
      =     L 8.3;
      BLD   103;
      A     DIX [AR2,P#40.4];
      =     L 8.4;
      BLD   103;
      A     DIX [AR2,P#41.5];
      =     L 8.5;
      BLD   103;
      A     DIX [AR2,P#42.0];
      =     L 8.6;
      BLD   103;
      A     DIX [AR2,P#42.1];
      =     L 8.7;
      BLD   103;
      A     DIX [AR2,P#42.2];
      =     L 9.0;
      BLD   103;
      A     "Always0";
      =     L 9.1;
      BLD   103;
      A     "Always0";
      =     L 9.2;
      BLD   103;
      A     "Always0";
      =     L 9.3;
      BLD   103;
      A     "Always0";
      =     L 9.4;
      BLD   103;
      A     "Always0";
      =     L 9.5;
      BLD   103;
      A     "Always0";
      =     L 9.6;
      BLD   103;
      AN    DIX [AR2,P#44.1];
      =     L 9.7;
      BLD   103;
      CALL  "HF3_B_T_W_FC51" (
           Bit_0                    := L 8.0,
           Bit_1                    := L 8.1,
           Bit_2                    := L 8.2,
           Bit_3                    := L 8.3,
           Bit_4                    := L 8.4,
           Bit_5                    := L 8.5,
           Bit_6                    := L 8.6,
           Bit_7                    := L 8.7,
           Bit_8                    := L 9.0,
           Bit_9                    := L 9.1,
           Bit_10                   := L 9.2,
           Bit_11                   := L 9.3,
           Bit_12                   := L 9.4,
           Bit_13                   := L 9.5,
           Bit_14                   := L 9.6,
           Bit_15                   := L 9.7,
           Word1                    := #ToHMI);
      NOP   0;
NETWORK
TITLE = 结束功能块
      SET;
      SAVE;
      CLR;
      BEU;
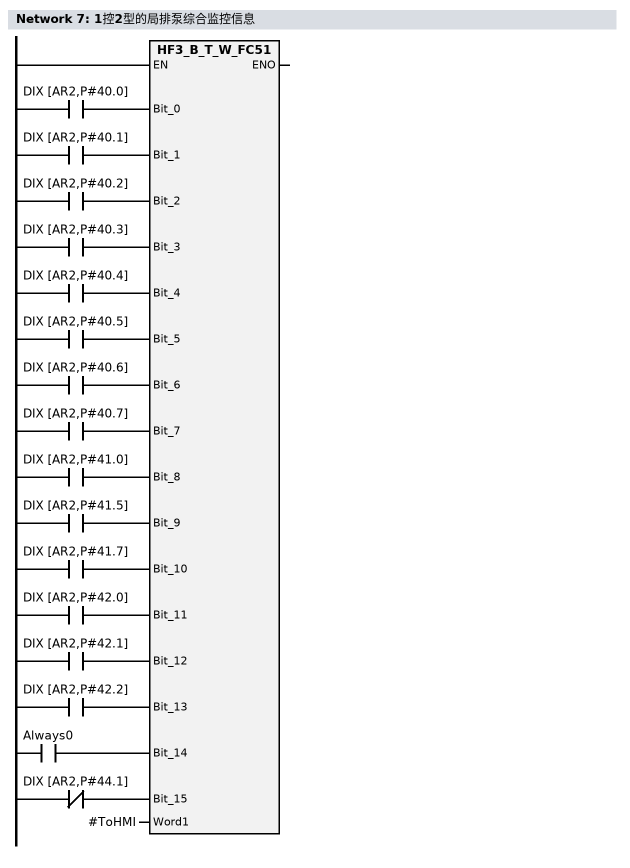
NETWORK
TITLE = 1控2型的局排泵综合监控信息
PUM2: A     DIX [AR2,P#40.0];
      =     L 8.0;
      BLD   103;
      A     DIX [AR2,P#40.1];
      =     L 8.1;
      BLD   103;
      A     DIX [AR2,P#40.2];
      =     L 8.2;
      BLD   103;
      A     DIX [AR2,P#40.3];
      =     L 8.3;
      BLD   103;
      A     DIX [AR2,P#40.4];
      =     L 8.4;
      BLD   103;
      A     DIX [AR2,P#40.5];
      =     L 8.5;
      BLD   103;
      A     DIX [AR2,P#40.6];
      =     L 8.6;
      BLD   103;
      A     DIX [AR2,P#40.7];
      =     L 8.7;
      BLD   103;
      A     DIX [AR2,P#41.0];
      =     L 9.0;
      BLD   103;
      A     DIX [AR2,P#41.5];
      =     L 9.1;
      BLD   103;
      A     DIX [AR2,P#41.7];
      =     L 9.2;
      BLD   103;
      A     DIX [AR2,P#42.0];
      =     L 9.3;
      BLD   103;
      A     DIX [AR2,P#42.1];
      =     L 9.4;
      BLD   103;
      A     DIX [AR2,P#42.2];
      =     L 9.5;
      BLD   103;
      A     "Always0";
      =     L 9.6;
      BLD   103;
      AN    DIX [AR2,P#44.1];
      =     L 9.7;
      BLD   103;
      CALL  "HF3_B_T_W_FC51" (
           Bit_0                    := L 8.0,
           Bit_1                    := L 8.1,
           Bit_2                    := L 8.2,
           Bit_3                    := L 8.3,
           Bit_4                    := L 8.4,
           Bit_5                    := L 8.5,
           Bit_6                    := L 8.6,
           Bit_7                    := L 8.7,
           Bit_8                    := L 9.0,
           Bit_9                    := L 9.1,
           Bit_10                   := L 9.2,
           Bit_11                   := L 9.3,
           Bit_12                   := L 9.4,
           Bit_13                   := L 9.5,
           Bit_14                   := L 9.6,
           Bit_15                   := L 9.7,
           Word1                    := #ToHMI);
      NOP   0;
NETWORK
TITLE = 结束功能块
      SET;
      SAVE;
      CLR;
      BEU;
END_FUNCTION_BLOCK

FUNCTION_BLOCK "HF3_UPS_FB2611"	// FB 2611
VERSION : 0.1
VAR
  UPS : FB 2612;
END_VAR
BEGIN
NETWORK
TITLE = UPS
// (network holds code this reader does not know; not shown)
END_FUNCTION_BLOCK

FUNCTION_BLOCK "HF3_UPS_FB2612"	// FB 2612
TITLE = UPS Status
//
//UPS Status Obtain
//
AUTHOR : SUNWIN_G
FAMILY : SUNWIN
NAME : UPS_Read
VERSION : 1.0
VAR_INPUT
  DB_NO : INT ;
END_VAR
VAR_OUTPUT
  AI_Status : ARRAY  [0 .. 11 ] OF INT ;
  DI_Status : WORD ;
END_VAR
VAR
  I : INT ;
  J : INT ;
  BOOL_Arr : ARRAY  [0 .. 15 ] OF BOOL ;
END_VAR
BEGIN
// body was compiled from an SCL source; compiled code not shown
END_FUNCTION_BLOCK

FUNCTION_BLOCK "HF3_DT_FB2621"	// FB 2621
VERSION : 0.1
VAR
  H420_02_K : FB 2622;
END_VAR
BEGIN
NETWORK
TITLE = H420_02_K
      BLD   14;
      =     L 7.0;
      L     DINO;
      T     LW 5;
      CDB;
      OPN   DI [LW 5];
      TAR2  LD 1;
      +AR2  P#0.0;
      UC    "HF3_DT_FB2622";
      LAR2  LD 1;
      L     #H420_02_K.ToHMI;
      OPN   DI 6004;
      T     DIW 702;
      OPN   DI [LW 5];
      L     #H420_02_K.Floor;
      OPN   DI 6004;
      T     DIW 704;
      OPN   DI [LW 5];
      CDB;
      BLD   15;
      NOP   0;
END_FUNCTION_BLOCK

FUNCTION_BLOCK "HF3_DT_FB2622"	// FB 2622
VERSION : 0.1
VAR_INPUT
  DB_NO : INT ;
  Multi : BOOL ;	//是否有多个水泵并线
  in_stradr : INT ;	//读命令状态开始地址
END_VAR
VAR_OUTPUT
  ToHMI : WORD ;
  Floor : WORD ;
END_VAR
VAR
  IN_RD1 : WORD ;
  COMM_HB : WORD ;
  floor_temp : WORD ;
  inRD_Temp : ARRAY  [0 .. 15 ] OF BOOL ;
  CommOK_Temp : BOOL ;	//通信状态中间变量
  CommOK : BOOL ;
  TON1 : SFB 4;
END_VAR
VAR_TEMP
  DI_reg : INT ;	//instance DB号
  db_no_temp : INT ;
  AR2_VALUE : DWORD ;	//AR2寄存器原始值
END_VAR
BEGIN
NETWORK
TITLE =
      CLR;
      L     #DB_NO;
      T     #db_no_temp;
//当CP340接入多个垂梯时
      L     P#0.0;
      LAR1;
      A     #Multi;
      JCN   sigl;
      L     #in_stradr;
      SLD   3;
      LAR1;
// 寄存器40001 、40002内容传递 通讯状态传递
sigl: OPN   DB [#db_no_temp];	//寄存器40001内容传递     DI状态
// DI״̬
      L     DBW [AR1,P#2.0];
      T     #IN_RD1;	//传递至IN_RD1内   
//电梯楼层
      L     DBW [AR1,P#4.0];	//寄存器40002内容传递 楼层信息
      T     #floor_temp;	//传递至 floor_temp
//通信状态判断
      L     DBW [AR1,P#0.0];
      T     #COMM_HB;	//该设备通讯状态   0为正常
//楼层值传递
      L     #floor_temp;
      AW    W#16#7;
      T     #Floor;
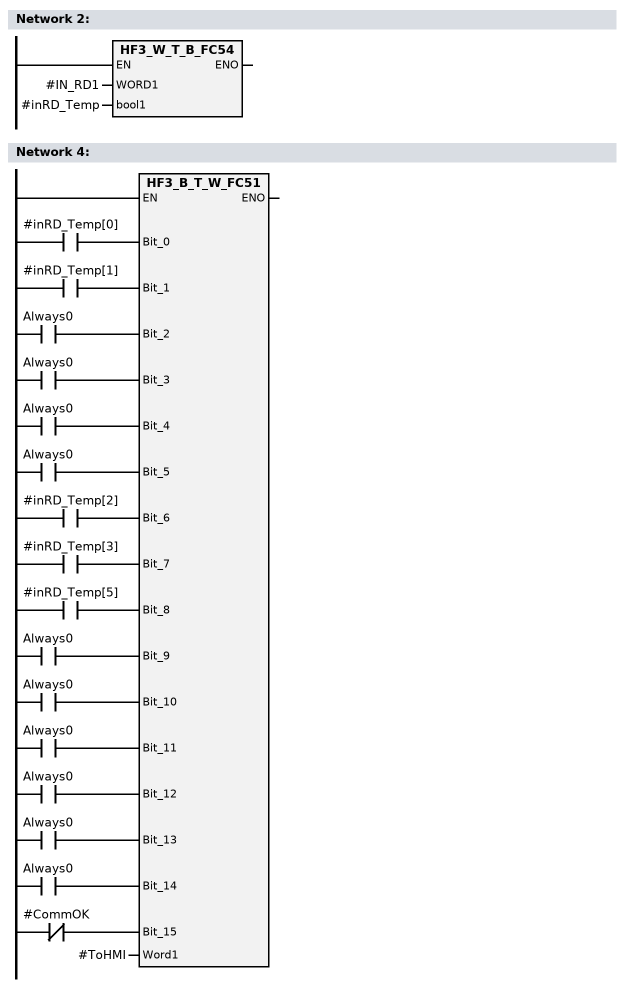
NETWORK
TITLE =
//  L     #inRD_Floor
//T     #Floor
//NOP   0
      CALL  "HF3_W_T_B_FC54" (
           WORD1                    := #IN_RD1,
           bool1                    := #inRD_Temp);
      NOP   0;
NETWORK
TITLE =
      CLR;
      L     #COMM_HB;
      L     W#16#0;
      <>I;
      =     #CommOK_Temp;
      BLD   16;
      =     L 14.0;
      L     DINO;
      T     LW 12;
      CDB;
      OPN   DI [LW 12];
      TAR2  LD 8;
      A     DBX [AR2,P#18.0];
      =     DIX [AR2,P#20.0];
      L     L#3000;
      T     DID [AR2,P#22.0];
      +AR2  P#20.0;
      UC    "TON";
      LAR2  LD 8;
      A     DIX [AR2,P#26.0];
      =     DBX [AR2,P#18.1];
      CDB;
      BLD   17;
NETWORK
TITLE =
      A     #inRD_Temp[0];
      =     L 8.0;
      BLD   103;
      A     #inRD_Temp[1];
      =     L 8.1;
      BLD   103;
      A     "Always0";
      =     L 8.2;
      BLD   103;
      A     "Always0";
      =     L 8.3;
      BLD   103;
      A     "Always0";
      =     L 8.4;
      BLD   103;
      A     "Always0";
      =     L 8.5;
      BLD   103;
      A     #inRD_Temp[2];
      =     L 8.6;
      BLD   103;
      A     #inRD_Temp[3];
      =     L 8.7;
      BLD   103;
      A     #inRD_Temp[5];
      =     L 9.0;
      BLD   103;
      A     "Always0";
      =     L 9.1;
      BLD   103;
      A     "Always0";
      =     L 9.2;
      BLD   103;
      A     "Always0";
      =     L 9.3;
      BLD   103;
      A     "Always0";
      =     L 9.4;
      BLD   103;
      A     "Always0";
      =     L 9.5;
      BLD   103;
      A     "Always0";
      =     L 9.6;
      BLD   103;
      AN    #CommOK;
      =     L 9.7;
      BLD   103;
      CALL  "HF3_B_T_W_FC51" (
           Bit_0                    := L 8.0,
           Bit_1                    := L 8.1,
           Bit_2                    := L 8.2,
           Bit_3                    := L 8.3,
           Bit_4                    := L 8.4,
           Bit_5                    := L 8.5,
           Bit_6                    := L 8.6,
           Bit_7                    := L 8.7,
           Bit_8                    := L 9.0,
           Bit_9                    := L 9.1,
           Bit_10                   := L 9.2,
           Bit_11                   := L 9.3,
           Bit_12                   := L 9.4,
           Bit_13                   := L 9.5,
           Bit_14                   := L 9.6,
           Bit_15                   := L 9.7,
           Word1                    := #ToHMI);
      NOP   0;
END_FUNCTION_BLOCK

FUNCTION_BLOCK "HF3_FT_FB2631"	// FB 2631
VERSION : 0.1
VAR
  E325_02_N : FB 2632;
  E325_01_N : FB 2632;
  E420_01_N : FB 2632;
  E420_05_K : FB 2632;
  E420_06_K : FB 2632;
  E420_07_K : FB 2632;
END_VAR
BEGIN
NETWORK
TITLE = E420_01_N
      A     "Always0";
      =     L 0.0;
      BLD   103;
      BLD   14;
      =     L 7.0;
      L     DINO;
      T     LW 5;
      CDB;
      OPN   DI [LW 5];
      TAR2  LD 1;
      L     2105;
      T     DIW [AR2,P#84.0];
      A     L 0.0;
      =     DIX [AR2,P#86.0];
      L     0;
      T     DIW [AR2,P#88.0];
      +AR2  P#84.0;
      UC    "HF4_FT_FB2362";
      LAR2  LD 1;
      L     DIW [AR2,P#90.0];
      OPN   DI 6004;
      T     DIW 690;
      OPN   DI [LW 5];
      CDB;
      BLD   15;
      NOP   0;
NETWORK
TITLE = E420_05_K
      A     "Always0";
      =     L 0.0;
      BLD   103;
      BLD   14;
      =     L 7.0;
      L     DINO;
      T     LW 5;
      CDB;
      OPN   DI [LW 5];
      TAR2  LD 1;
      L     2065;
      T     DIW [AR2,P#126.0];
      A     L 0.0;
      =     DIX [AR2,P#128.0];
      +AR2  P#126.0;
      UC    "HF4_FT_FB2362";
      LAR2  LD 1;
      L     DIW [AR2,P#132.0];
      OPN   DI 6004;
      T     DIW 692;
      OPN   DI [LW 5];
      CDB;
      BLD   15;
      NOP   0;
NETWORK
TITLE = E420_06_K
      A     "Always1";
      =     L 0.0;
      BLD   103;
      BLD   14;
      =     L 7.0;
      L     DINO;
      T     LW 5;
      CDB;
      OPN   DI [LW 5];
      TAR2  LD 1;
      L     2105;
      T     DIW [AR2,P#168.0];
      A     L 0.0;
      =     DIX [AR2,P#170.0];
      L     0;
      T     DIW [AR2,P#172.0];
      +AR2  P#168.0;
      UC    "HF4_FT_FB2362";
      LAR2  LD 1;
      L     DIW [AR2,P#174.0];
      OPN   DI 6004;
      T     DIW 694;
      OPN   DI [LW 5];
      CDB;
      BLD   15;
      NOP   0;
NETWORK
TITLE = E420_07_K
      A     "Always1";
      =     L 0.0;
      BLD   103;
      BLD   14;
      =     L 7.0;
      L     DINO;
      T     LW 5;
      CDB;
      OPN   DI [LW 5];
      TAR2  LD 1;
      L     2105;
      T     DIW [AR2,P#210.0];
      A     L 0.0;
      =     DIX [AR2,P#212.0];
      L     8;
      T     DIW [AR2,P#214.0];
      +AR2  P#210.0;
      UC    "HF4_FT_FB2362";
      LAR2  LD 1;
      L     DIW [AR2,P#216.0];
      OPN   DI 6004;
      T     DIW 696;
      OPN   DI [LW 5];
      CDB;
      BLD   15;
      NOP   0;
END_FUNCTION_BLOCK

FUNCTION_BLOCK "HF4_FT_FB2362"	// FB 2632
VERSION : 0.1
VAR_INPUT
  DB_NO : INT ;
  Multi : BOOL ;	//是否有多个水泵并线
  in_stradr : INT ;	//读命令状态开始地址
END_VAR
VAR_OUTPUT
  ToHMI : WORD ;
END_VAR
VAR
  IN_RD1 : WORD ;
  IN_RD2 : WORD ;
  COMM_HB : WORD ;
  inRD_Temp1 : ARRAY  [0 .. 15 ] OF BOOL ;
  inRD_Temp2 : ARRAY  [0 .. 15 ] OF BOOL ;
  CommOK_Temp : BOOL ;
  CommOK : BOOL ;
  TON1 : SFB 4;
END_VAR
VAR_TEMP
  DI_reg : INT ;	//instance DB号
  db_no_temp : INT ;
  AR2_VALUE : DWORD ;	//AR2寄存器原始值
END_VAR
BEGIN
NETWORK
TITLE = 状态读取
      CLR;
      L     #DB_NO;
      T     #db_no_temp;
//当CP340接入多个扶梯时
      L     P#0.0;
      LAR1;
      A     #Multi;
      JCN   sigl;
      L     #in_stradr;
      SLD   3;
      LAR1;
// 寄存器400022 、40021内容传递 通讯状态传递       厂家点表错误
sigl: OPN   DB [#db_no_temp];
// DI״̬
      L     DBW [AR1,P#4.0];	//寄存器400022内容传递 DI状态 
      T     #IN_RD1;	//传递至IN_RD1内   
//读40002 40021由两条读命令实现 读取偏移位加2
      L     DBW [AR1,P#2.0];	//寄存器40021内容传递 DI状态 
      T     #IN_RD2;	//传递至IN_RD2内   
//通信状态判断
      L     DBW [AR1,P#0.0];
      T     #COMM_HB;	//该设备通讯状态   0为正常
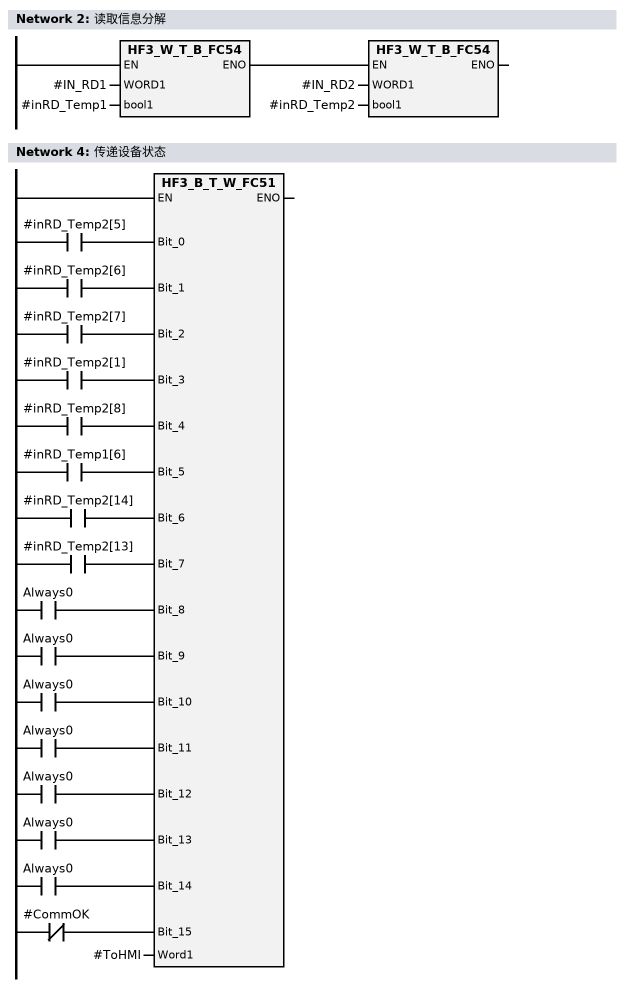
NETWORK
TITLE = 读取信息分解
      A(;
      CALL  "HF3_W_T_B_FC54" (
           WORD1                    := #IN_RD1,
           bool1                    := #inRD_Temp1);
      A     BR;
      );
      JNB   _001;
      CALL  "HF3_W_T_B_FC54" (
           WORD1                    := #IN_RD2,
           bool1                    := #inRD_Temp2);
_001: NOP   0;
NETWORK
TITLE = 通讯状态判断
      CLR;
      L     #COMM_HB;
      L     W#16#0;
      <>I;
      =     #CommOK_Temp;
      BLD   16;
      =     L 14.0;
      L     DINO;
      T     LW 12;
      CDB;
      OPN   DI [LW 12];
      TAR2  LD 8;
      A     DBX [AR2,P#18.0];
      =     DIX [AR2,P#20.0];
      L     L#3000;
      T     DID [AR2,P#22.0];
      +AR2  P#20.0;
      UC    "TON";
      LAR2  LD 8;
      A     DIX [AR2,P#26.0];
      =     DBX [AR2,P#18.1];
      CDB;
      BLD   17;
NETWORK
TITLE = 传递设备状态
//4.7修改寄存器对应偏移位
      A     #inRD_Temp2[5];
      =     L 8.0;
      BLD   103;
      A     #inRD_Temp2[6];
      =     L 8.1;
      BLD   103;
      A     #inRD_Temp2[7];
      =     L 8.2;
      BLD   103;
      A     #inRD_Temp2[1];
      =     L 8.3;
      BLD   103;
      A     #inRD_Temp2[8];
      =     L 8.4;
      BLD   103;
      A     #inRD_Temp1[6];
      =     L 8.5;
      BLD   103;
      A     #inRD_Temp2[14];
      =     L 8.6;
      BLD   103;
      A     #inRD_Temp2[13];
      =     L 8.7;
      BLD   103;
      A     "Always0";
      =     L 9.0;
      BLD   103;
      A     "Always0";
      =     L 9.1;
      BLD   103;
      A     "Always0";
      =     L 9.2;
      BLD   103;
      A     "Always0";
      =     L 9.3;
      BLD   103;
      A     "Always0";
      =     L 9.4;
      BLD   103;
      A     "Always0";
      =     L 9.5;
      BLD   103;
      A     "Always0";
      =     L 9.6;
      BLD   103;
      AN    #CommOK;
      =     L 9.7;
      BLD   103;
      CALL  "HF3_B_T_W_FC51" (
           Bit_0                    := L 8.0,
           Bit_1                    := L 8.1,
           Bit_2                    := L 8.2,
           Bit_3                    := L 8.3,
           Bit_4                    := L 8.4,
           Bit_5                    := L 8.5,
           Bit_6                    := L 8.6,
           Bit_7                    := L 8.7,
           Bit_8                    := L 9.0,
           Bit_9                    := L 9.1,
           Bit_10                   := L 9.2,
           Bit_11                   := L 9.3,
           Bit_12                   := L 9.4,
           Bit_13                   := L 9.5,
           Bit_14                   := L 9.6,
           Bit_15                   := L 9.7,
           Word1                    := #ToHMI);
      NOP   0;
END_FUNCTION_BLOCK

FUNCTION_BLOCK "HF3_IMCC_TVF_FB2651"	// FB 2651
TITLE = IMCCϵͳTVF_A1
VERSION : 0.1
VAR
  TVF_A1 : FB 2652;
  TVF_A2 : FB 2652;
  PT : TIME  := T#45S;
END_VAR
BEGIN
NETWORK
TITLE = 隧道风机TVF_A1
      A     "Always0";
      =     L 0.0;
      BLD   103;
      A     "Always1";
      =     L 0.1;
      BLD   103;
      A     "Maste_To_Slave_Mod_DB".FireAlarm;
      =     L 0.2;
      BLD   103;
      A     "Maste_To_Slave_Mod_DB".BlockAlarm;
      =     L 0.3;
      BLD   103;
      BLD   14;
      =     L 7.0;
      L     DINO;
      T     LW 5;
      CDB;
      OPN   DI [LW 5];
      TAR2  LD 1;
      A     L 0.0;
      =     #TVF_A1.Main;
      BLD   11;
      L     W#16#1002;
      T     LW 10;
      L     28;
      T     LW 12;
      L     2291;
      T     LW 14;
      L     P#DBX 356.0;
      T     LD 16;
      L     W#16#1002;
      T     LW 20;
      L     28;
      T     LW 22;
      L     DINO;
      T     LW 24;
      +AR2  P#2.0;
      TAR2;
      LAR2  LD 1;
      T     LD 26;
      UC    "BLKMOV";
      {     P#L 10.0, P#L 8.0, P#L 20.0 };
      L     394;
      T     #TVF_A1.HMI_Adr;
      OPN   DI 6040;
      L     DIW 80;
      OPN   DI [LW 5];
      T     #TVF_A1.SCtrl;
      BLD   11;
      L     W#16#1002;
      T     LW 10;
      L     2;
      T     LW 12;
      L     7004;
      T     LW 14;
      L     P#DBX 16.0;
      T     LD 16;
      L     W#16#1002;
      T     LW 20;
      L     2;
      T     LW 22;
      L     DINO;
      T     LW 24;
      +AR2  P#34.0;
      TAR2;
      LAR2  LD 1;
      T     LD 26;
      UC    "BLKMOV";
      {     P#L 10.0, P#L 8.0, P#L 20.0 };
      BLD   11;
      L     W#16#1002;
      T     LW 10;
      L     2;
      T     LW 12;
      L     7005;
      T     LW 14;
      L     P#DBX 2.0;
      T     LD 16;
      L     W#16#1002;
      T     LW 20;
      L     2;
      T     LW 22;
      L     DINO;
      T     LW 24;
      +AR2  P#36.0;
      TAR2;
      LAR2  LD 1;
      T     LD 26;
      UC    "BLKMOV";
      {     P#L 10.0, P#L 8.0, P#L 20.0 };
      A     L 0.1;
      =     #TVF_A1.Open;
      L     DBD [AR2,P#384.0];
      T     #TVF_A1.PT01;
      BLD   11;
      L     W#16#1002;
      T     LW 10;
      L     2;
      T     LW 12;
      L     7005;
      T     LW 14;
      L     P#DBX 32.0;
      T     LD 16;
      L     W#16#1002;
      T     LW 20;
      L     2;
      T     LW 22;
      L     DINO;
      T     LW 24;
      +AR2  P#44.0;
      TAR2;
      LAR2  LD 1;
      T     LD 26;
      UC    "BLKMOV";
      {     P#L 10.0, P#L 8.0, P#L 20.0 };
      OPN   DI 7005;
      L     DIW 312;
      OPN   DI [LW 5];
      T     #TVF_A1.H_P_All_Ctrl;
      A     L 0.2;
      =     #TVF_A1.FireAlarm;
      A     L 0.3;
      =     #TVF_A1.BlockAlarm;
      +AR2  P#0.0;
      UC    "HF4_IMCC_TVF_FB2652";
      LAR2  LD 1;
      L     #TVF_A1.qtWR;
      OPN   DI 2292;
      T     DIW 92;
      OPN   DI [LW 5];
      L     #TVF_A1.RT;
      OPN   DI 6004;
      T     DID 424;
      OPN   DI [LW 5];
      L     #TVF_A1.SumFlt;
      OPN   DI 6004;
      T     DIW 428;
      OPN   DI [LW 5];
      A     #TVF_A1.Refuse;
      OPN   DI 7006;
      =     DIX 2.7;
      OPN   DI [LW 5];
      CDB;
      BLD   15;
      NOP   0;
NETWORK
TITLE = TVF_A2
      A     "Always0";
      =     L 0.0;
      BLD   103;
      A     "Always1";
      =     L 0.1;
      BLD   103;
      A     "Maste_To_Slave_Mod_DB".FireAlarm;
      =     L 0.2;
      BLD   103;
      A     "Maste_To_Slave_Mod_DB".BlockAlarm;
      =     L 0.3;
      BLD   103;
      BLD   14;
      =     L 7.0;
      L     DINO;
      T     LW 5;
      CDB;
      OPN   DI [LW 5];
      TAR2  LD 1;
      A     L 0.0;
      =     DIX [AR2,P#192.0];
      BLD   11;
      L     W#16#1002;
      T     LW 10;
      L     28;
      T     LW 12;
      L     2291;
      T     LW 14;
      L     P#DBX 384.0;
      T     LD 16;
      L     W#16#1002;
      T     LW 20;
      L     28;
      T     LW 22;
      L     DINO;
      T     LW 24;
      +AR2  P#194.0;
      TAR2;
      LAR2  LD 1;
      T     LD 26;
      UC    "BLKMOV";
      {     P#L 10.0, P#L 8.0, P#L 20.0 };
      L     438;
      T     DIW [AR2,P#222.0];
      OPN   DI 6040;
      L     DIW 82;
      OPN   DI [LW 5];
      T     DIW [AR2,P#224.0];
      BLD   11;
      L     W#16#1002;
      T     LW 10;
      L     2;
      T     LW 12;
      L     7004;
      T     LW 14;
      L     P#DBX 18.0;
      T     LD 16;
      L     W#16#1002;
      T     LW 20;
      L     2;
      T     LW 22;
      L     DINO;
      T     LW 24;
      +AR2  P#226.0;
      TAR2;
      LAR2  LD 1;
      T     LD 26;
      UC    "BLKMOV";
      {     P#L 10.0, P#L 8.0, P#L 20.0 };
      BLD   11;
      L     W#16#1002;
      T     LW 10;
      L     2;
      T     LW 12;
      L     7005;
      T     LW 14;
      L     P#DBX 2.0;
      T     LD 16;
      L     W#16#1002;
      T     LW 20;
      L     2;
      T     LW 22;
      L     DINO;
      T     LW 24;
      +AR2  P#228.0;
      TAR2;
      LAR2  LD 1;
      T     LD 26;
      UC    "BLKMOV";
      {     P#L 10.0, P#L 8.0, P#L 20.0 };
      A     L 0.1;
      =     DIX [AR2,P#230.0];
      L     DBD [AR2,P#384.0];
      T     DID [AR2,P#232.0];
      BLD   11;
      L     W#16#1002;
      T     LW 10;
      L     2;
      T     LW 12;
      L     7005;
      T     LW 14;
      L     P#DBX 32.0;
      T     LD 16;
      L     W#16#1002;
      T     LW 20;
      L     2;
      T     LW 22;
      L     DINO;
      T     LW 24;
      +AR2  P#236.0;
      TAR2;
      LAR2  LD 1;
      T     LD 26;
      UC    "BLKMOV";
      {     P#L 10.0, P#L 8.0, P#L 20.0 };
      OPN   DI 7005;
      L     DIW 312;
      OPN   DI [LW 5];
      T     DIW [AR2,P#238.0];
      A     L 0.2;
      =     DIX [AR2,P#240.0];
      A     L 0.3;
      =     DIX [AR2,P#240.1];
      +AR2  P#192.0;
      UC    "HF4_IMCC_TVF_FB2652";
      LAR2  LD 1;
      L     DIW [AR2,P#242.0];
      OPN   DI 2292;
      T     DIW 94;
      OPN   DI [LW 5];
      L     DID [AR2,P#244.0];
      OPN   DI 6004;
      T     DID 468;
      OPN   DI [LW 5];
      L     DIW [AR2,P#248.0];
      OPN   DI 6004;
      T     DIW 472;
      OPN   DI [LW 5];
      A     DIX [AR2,P#252.0];
      OPN   DI 7006;
      =     DIX 3.0;
      OPN   DI [LW 5];
      CDB;
      BLD   15;
      NOP   0;
END_FUNCTION_BLOCK

FUNCTION_BLOCK "HF4_IMCC_TVF_FB2652"	// FB 2652
VERSION : 0.1
VAR_INPUT
  Main : BOOL ;	//1:大端 2：小端
  IN_RD : ARRAY  [0 .. 13 ] OF WORD ;
  HMI_Adr : INT ;
  SCtrl : WORD ;	//上位控制命令
  MCtrl : ARRAY  [0 .. 3 ] OF //0-正转1-反转2-停止
  BOOL ;
  Mode : ARRAY  [0 .. 15 ] OF //0-模式开始1-结束2-执行中
  BOOL ;
  Open : BOOL ;	//连锁风阀开
  PT01 : TIME ;	//风机延时时间
  ALL : ARRAY  [0 .. 15 ] OF //0-单控1-模控2-时间表
  BOOL ;
  H_P_All_Ctrl : WORD ;
  FireAlarm : BOOL ;	//火灾信号
  BlockAlarm : BOOL ;	//阻塞信号
END_VAR
VAR_OUTPUT
  qtWR : WORD ;
  RT : REAL ;
  SumFlt : INT ;
  SumRun : INT ;
  Refuse : BOOL ;	//模式不符
  Stop : BOOL ;	//风机控制
END_VAR
VAR
  IN_RD1 : WORD ;
  qtWR_1 : WORD ;
  TOHMI_1 : WORD ;
  TOHMI_2 : WORD ;
  qtwr_temp : WORD ;
  DI_Temp1 : ARRAY  [0 .. 15 ] OF //设备状态字1
  BOOL ;
  DI_Temp2 : ARRAY  [0 .. 15 ] OF //设备状态字2
  BOOL ;
  DO_Temp : ARRAY  [0 .. 15 ] OF //输出状态字
  BOOL ;
  Ctrl : ARRAY  [0 .. 15 ] OF //0-正传1-反转2-停止
  BOOL ;
  SCtrl_Temp : ARRAY  [0 .. 15 ] OF //上位控制中间变量
  BOOL ;
  Latch : ARRAY  [0 .. 15 ] OF BOOL ;
  H_P_All_Ctrl_Temp : ARRAY  [0 .. 15 ] OF BOOL ;
  SFlag : BOOL ;	//单控标志
  McFlag : BOOL ;	//检修牌
  SingTout : BOOL ;	//单控超时
  QTout : BOOL ;	//输出超时
  Timeout : BOOL ;	//设备动作超时
  Flt : BOOL ;	//设备控制综合故障
  Ton1 : SFB 4;
  Ton2 : SFB 4;
  Ton3 : SFB 4;
  Ton4 : SFB 4;
  RunFaultSum : FB 2006;
END_VAR
VAR_TEMP
  AR2_Value : DWORD ;
  DI_NO : INT ;
  Data_Len : INT ;
  DB_NO : INT ;
END_VAR
BEGIN
NETWORK
TITLE =
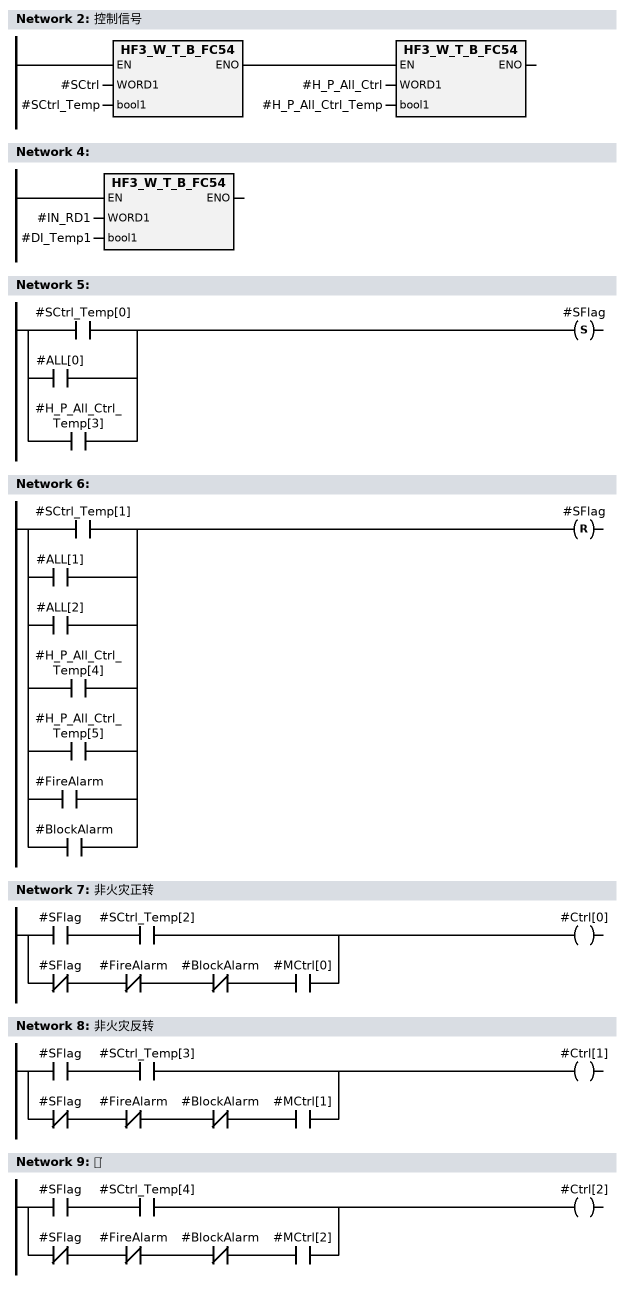
NETWORK
TITLE = 控制信号
      A(;
      CALL  "HF3_W_T_B_FC54" (
           WORD1                    := #SCtrl,
           bool1                    := #SCtrl_Temp);
      A     BR;
      );
      JNB   _001;
      CALL  "HF3_W_T_B_FC54" (
           WORD1                    := #H_P_All_Ctrl,
           bool1                    := #H_P_All_Ctrl_Temp);
_001: NOP   0;
NETWORK
TITLE = 初始化
////*5.18新更新,取消通讯故障
////*5.11新更新，所有数字量信息集中于第一个字中，第十五位为通讯故障
//第1个字BIT 0BAS
//第1个字BIT 1就地
//第1个字BIT 2正转运行状态
//第1个字BIT 3反转运行状态
//第1个字BIT 4风机停止状态
//第1个字BIT 5软启动故障
//第1个字BIT 6振动超高报警
//第1个字BIT 7轴承温度报警
//第1个字BIT 8绕组温度报警
//第1个字BIT 9电动机缺相
//第1个字BIT 10火灾切除保护信息
//第1个字BIT 11电动机过载
//
//
//
//
//第2个字电动机电流A
//第3个字电动机电流B
//第4个字电动机电流C
//第5个字电动机电压A
//第6个字电动机电压B
//第7个字电动机电压C
//第8个字前轴承温度
//第9个字后轴承温度
//第10个字绕组温度A
//第11个字绕组温度B
//第12个字绕组温度C
//第13个字水平振动
//第14个字垂直振动
//
      TAR2;
      T     #AR2_Value;
      L     6002;
      T     #DB_NO;
      A     #Main;	//此端是否为大端
      JC    big;
      L     6004;
      T     #DB_NO;
big:  L     DINO;	//存储背景数据块号
      T     #DI_NO;
      OPN   DB [#DB_NO];	//打开
      L     #HMI_Adr;
      SLD   3;
      LAR1;
// *********************事故风机中DI状态读取**********************
      L     #IN_RD[0];	//第一个字中包含数字量信息
      T     #IN_RD1;
//初始化AR2寄存器用于AI量传递
      TAR2;
      AD    DW#16#FFFFFF;
      L     P##IN_RD;
      +D;
      OD    DW#16#85000000;
      LAR2;
//*********************事故风机中AI状态读取**********************
//读取模拟量输入
      L     13;
ilop: T     #Data_Len;
      L     W [AR2,P#2.0];	//智能低压点表新更新，第二个字开始为模拟量
      T     DBW [AR1,P#4.0];
      +AR1  P#2.0;
      +AR2  P#2.0;
      L     #Data_Len;
      LOOP  ilop;
//恢复AR2 DI寄存器
      L     #AR2_Value;
      LAR2;
//     OPN   DI [#DI_NO]
NETWORK
TITLE =
      CALL  "HF3_W_T_B_FC54" (
           WORD1                    := #IN_RD1,
           bool1                    := #DI_Temp1);
      NOP   0;
NETWORK
TITLE =
      O     #SCtrl_Temp[0];
      O     #ALL[0];
      O     #H_P_All_Ctrl_Temp[3];
      S     #SFlag;
NETWORK
TITLE =
      O     #SCtrl_Temp[1];
      O     #ALL[1];
      O     #ALL[2];
      O     #H_P_All_Ctrl_Temp[4];
      O     #H_P_All_Ctrl_Temp[5];
      O     #FireAlarm;
      O     #BlockAlarm;
      R     #SFlag;
NETWORK
TITLE = 非火灾正转
      A     #SFlag;
      A     #SCtrl_Temp[2];
      O;
      AN    #SFlag;
      AN    #FireAlarm;
      AN    #BlockAlarm;
      A     #MCtrl[0];
      =     #Ctrl[0];
NETWORK
TITLE = 非火灾反转
      A     #SFlag;
      A     #SCtrl_Temp[3];
      O;
      AN    #SFlag;
      AN    #FireAlarm;
      AN    #BlockAlarm;
      A     #MCtrl[1];
      =     #Ctrl[1];
NETWORK
TITLE = ֹͣ
      A     #SFlag;
      A     #SCtrl_Temp[4];
      O;
      AN    #SFlag;
      AN    #FireAlarm;
      AN    #BlockAlarm;
      A     #MCtrl[2];
      =     #Ctrl[2];
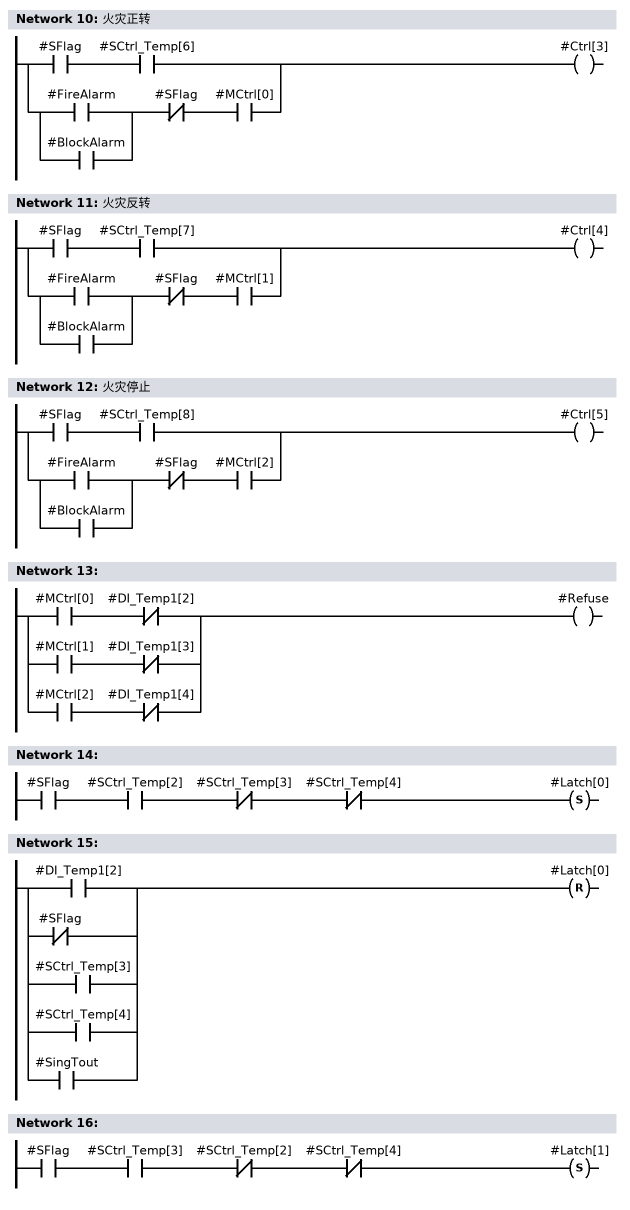
NETWORK
TITLE = 火灾正转
      A     #SFlag;
      A     #SCtrl_Temp[6];
      O;
      A(;
      O     #FireAlarm;
      O     #BlockAlarm;
      );
      AN    #SFlag;
      A     #MCtrl[0];
      =     #Ctrl[3];
NETWORK
TITLE = 火灾反转
      A     #SFlag;
      A     #SCtrl_Temp[7];
      O;
      A(;
      O     #FireAlarm;
      O     #BlockAlarm;
      );
      AN    #SFlag;
      A     #MCtrl[1];
      =     #Ctrl[4];
NETWORK
TITLE = 火灾停止
      A     #SFlag;
      A     #SCtrl_Temp[8];
      O;
      A(;
      O     #FireAlarm;
      O     #BlockAlarm;
      );
      AN    #SFlag;
      A     #MCtrl[2];
      =     #Ctrl[5];
NETWORK
TITLE =
      A     #MCtrl[0];
      AN    #DI_Temp1[2];
      O;
      A     #MCtrl[1];
      AN    #DI_Temp1[3];
      O;
      A     #MCtrl[2];
      AN    #DI_Temp1[4];
      =     #Refuse;
NETWORK
TITLE =
      A     #SFlag;
      A     #SCtrl_Temp[2];
      AN    #SCtrl_Temp[3];
      AN    #SCtrl_Temp[4];
      S     #Latch[0];
NETWORK
TITLE =
      O     #DI_Temp1[2];
      ON    #SFlag;
      O     #SCtrl_Temp[3];
      O     #SCtrl_Temp[4];
      O     #SingTout;
      R     #Latch[0];
NETWORK
TITLE =
      A     #SFlag;
      A     #SCtrl_Temp[3];
      AN    #SCtrl_Temp[2];
      AN    #SCtrl_Temp[4];
      S     #Latch[1];
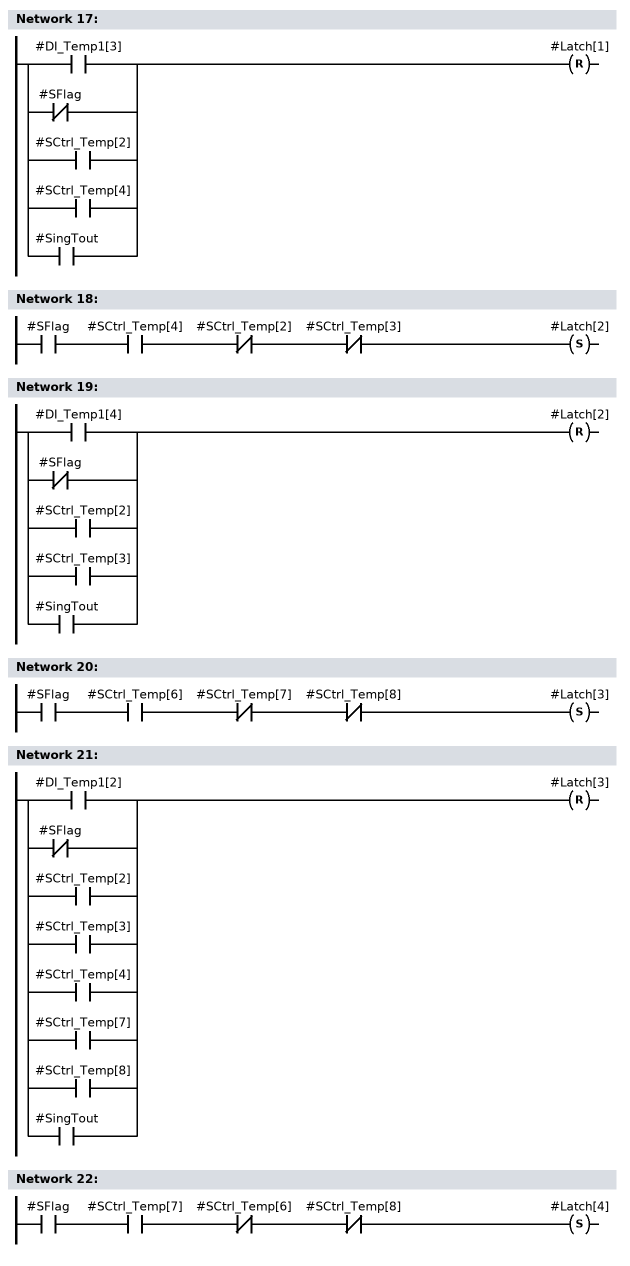
NETWORK
TITLE =
      O     #DI_Temp1[3];
      ON    #SFlag;
      O     #SCtrl_Temp[2];
      O     #SCtrl_Temp[4];
      O     #SingTout;
      R     #Latch[1];
NETWORK
TITLE =
      A     #SFlag;
      A     #SCtrl_Temp[4];
      AN    #SCtrl_Temp[2];
      AN    #SCtrl_Temp[3];
      S     #Latch[2];
NETWORK
TITLE =
      O     #DI_Temp1[4];
      ON    #SFlag;
      O     #SCtrl_Temp[2];
      O     #SCtrl_Temp[3];
      O     #SingTout;
      R     #Latch[2];
NETWORK
TITLE =
      A     #SFlag;
      A     #SCtrl_Temp[6];
      AN    #SCtrl_Temp[7];
      AN    #SCtrl_Temp[8];
      S     #Latch[3];
NETWORK
TITLE =
      O     #DI_Temp1[2];
      ON    #SFlag;
      O     #SCtrl_Temp[2];
      O     #SCtrl_Temp[3];
      O     #SCtrl_Temp[4];
      O     #SCtrl_Temp[7];
      O     #SCtrl_Temp[8];
      O     #SingTout;
      R     #Latch[3];
NETWORK
TITLE =
      A     #SFlag;
      A     #SCtrl_Temp[7];
      AN    #SCtrl_Temp[6];
      AN    #SCtrl_Temp[8];
      S     #Latch[4];
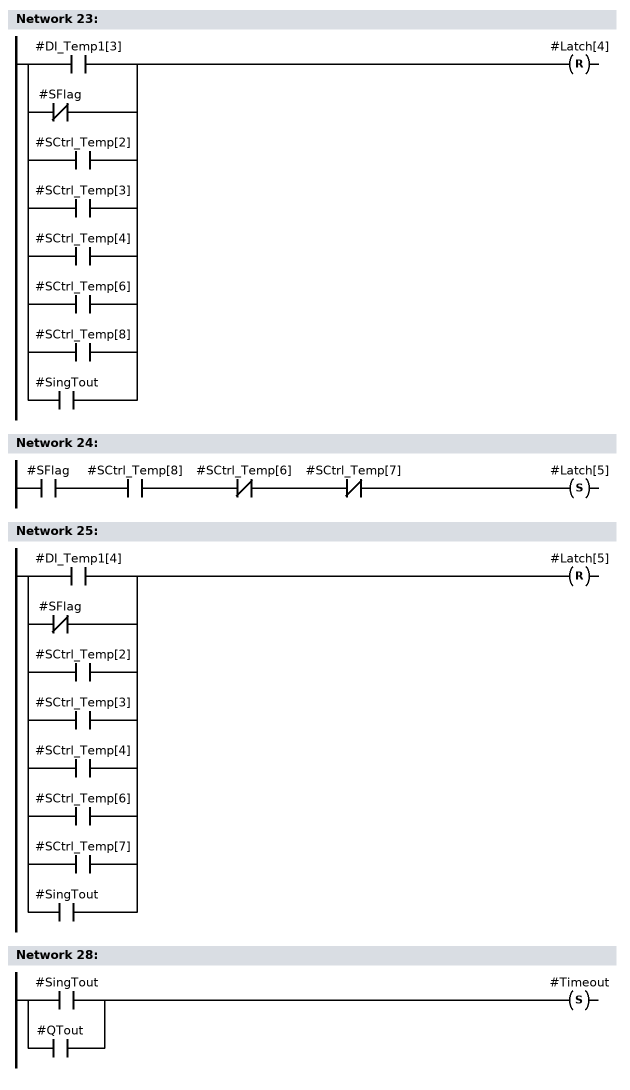
NETWORK
TITLE =
      O     #DI_Temp1[3];
      ON    #SFlag;
      O     #SCtrl_Temp[2];
      O     #SCtrl_Temp[3];
      O     #SCtrl_Temp[4];
      O     #SCtrl_Temp[6];
      O     #SCtrl_Temp[8];
      O     #SingTout;
      R     #Latch[4];
NETWORK
TITLE =
      A     #SFlag;
      A     #SCtrl_Temp[8];
      AN    #SCtrl_Temp[6];
      AN    #SCtrl_Temp[7];
      S     #Latch[5];
NETWORK
TITLE =
      O     #DI_Temp1[4];
      ON    #SFlag;
      O     #SCtrl_Temp[2];
      O     #SCtrl_Temp[3];
      O     #SCtrl_Temp[4];
      O     #SCtrl_Temp[6];
      O     #SCtrl_Temp[7];
      O     #SingTout;
      R     #Latch[5];
NETWORK
TITLE =
      A(;
      O     #Latch[0];
      O     #Latch[1];
      O     #Latch[2];
      O     #Latch[3];
      O     #Latch[4];
      O     #Latch[5];
      );
      =     L 10.0;
      BLD   103;
      BLD   16;
      =     L 17.0;
      L     DINO;
      T     LW 15;
      CDB;
      OPN   DI [LW 15];
      TAR2  LD 11;
      A     L 10.0;
      =     DIX [AR2,P#88.0];
      L     DBD [AR2,P#40.0];
      T     DID [AR2,P#90.0];
      +AR2  P#88.0;
      UC    "TON";
      LAR2  LD 11;
      A     DIX [AR2,P#94.0];
      =     DBX [AR2,P#86.2];
      CDB;
      BLD   17;
      NOP   0;
NETWORK
TITLE =
      A(;
      O     #DO_Temp[0];
      O     #DO_Temp[1];
      O     #DO_Temp[2];
      O     #DO_Temp[3];
      O     #DO_Temp[4];
      O     #DO_Temp[5];
      );
      =     L 10.0;
      BLD   103;
      BLD   16;
      =     L 17.0;
      L     DINO;
      T     LW 15;
      CDB;
      OPN   DI [LW 15];
      TAR2  LD 11;
      A     L 10.0;
      =     DIX [AR2,P#110.0];
      L     DBD [AR2,P#40.0];
      T     DID [AR2,P#112.0];
      +AR2  P#110.0;
      UC    "TON";
      LAR2  LD 11;
      A     DIX [AR2,P#116.0];
      =     DBX [AR2,P#86.3];
      CDB;
      BLD   17;
      NOP   0;
NETWORK
TITLE =
      O     #SingTout;
      O     #QTout;
      S     #Timeout;
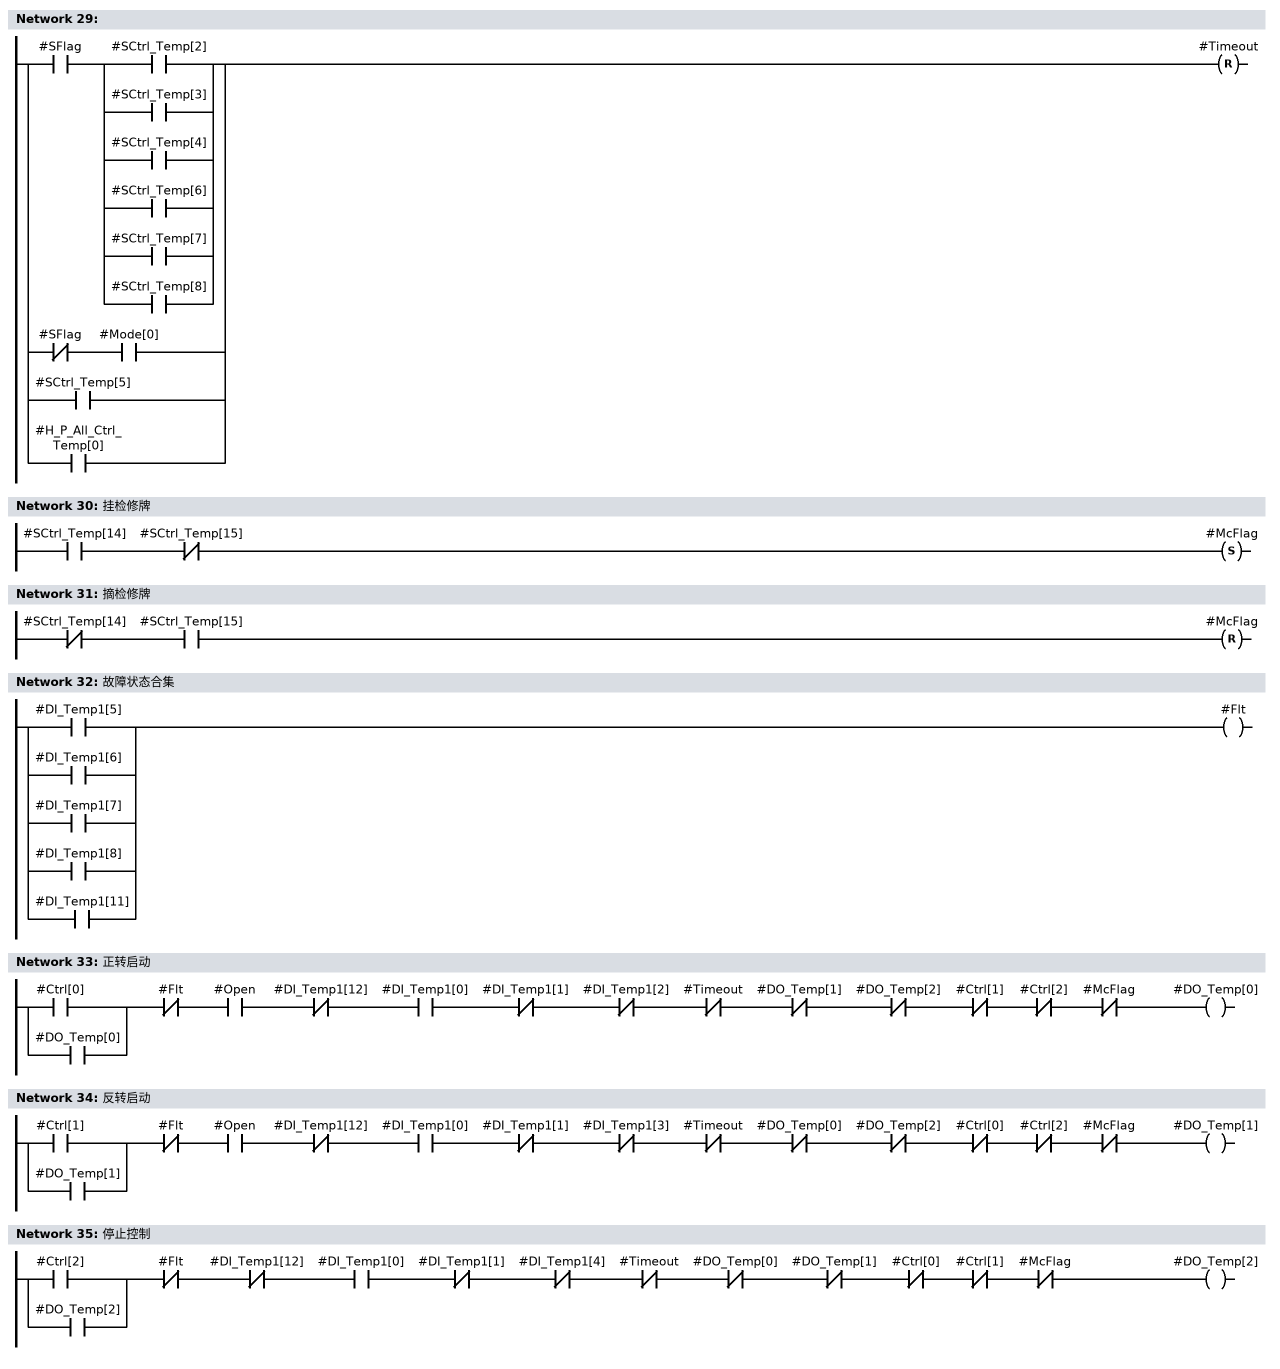
NETWORK
TITLE =
      A     #SFlag;
      A(;
      O     #SCtrl_Temp[2];
      O     #SCtrl_Temp[3];
      O     #SCtrl_Temp[4];
      O     #SCtrl_Temp[6];
      O     #SCtrl_Temp[7];
      O     #SCtrl_Temp[8];
      );
      O;
      AN    #SFlag;
      A     #Mode[0];
      O     #SCtrl_Temp[5];
      O     #H_P_All_Ctrl_Temp[0];
      R     #Timeout;
NETWORK
TITLE = 挂检修牌
      A     #SCtrl_Temp[14];
      AN    #SCtrl_Temp[15];
      S     #McFlag;
NETWORK
TITLE = 摘检修牌
      AN    #SCtrl_Temp[14];
      A     #SCtrl_Temp[15];
      R     #McFlag;
NETWORK
TITLE = 故障状态合集
      O     #DI_Temp1[5];
      O     #DI_Temp1[6];
      O     #DI_Temp1[7];
      O     #DI_Temp1[8];
      O     #DI_Temp1[11];
      =     #Flt;
NETWORK
TITLE = 正转启动
      A(;
      O     #Ctrl[0];
      O     #DO_Temp[0];
      );
      AN    #Flt;
      A     #Open;
      AN    #DI_Temp1[12];
      A     #DI_Temp1[0];
      AN    #DI_Temp1[1];
      AN    #DI_Temp1[2];
      AN    #Timeout;
      AN    #DO_Temp[1];
      AN    #DO_Temp[2];
      AN    #Ctrl[1];
      AN    #Ctrl[2];
      AN    #McFlag;
      =     #DO_Temp[0];
NETWORK
TITLE = 反转启动
      A(;
      O     #Ctrl[1];
      O     #DO_Temp[1];
      );
      AN    #Flt;
      A     #Open;
      AN    #DI_Temp1[12];
      A     #DI_Temp1[0];
      AN    #DI_Temp1[1];
      AN    #DI_Temp1[3];
      AN    #Timeout;
      AN    #DO_Temp[0];
      AN    #DO_Temp[2];
      AN    #Ctrl[0];
      AN    #Ctrl[2];
      AN    #McFlag;
      =     #DO_Temp[1];
NETWORK
TITLE = 停止控制
      A(;
      O     #Ctrl[2];
      O     #DO_Temp[2];
      );
      AN    #Flt;
      AN    #DI_Temp1[12];
      A     #DI_Temp1[0];
      AN    #DI_Temp1[1];
      AN    #DI_Temp1[4];
      AN    #Timeout;
      AN    #DO_Temp[0];
      AN    #DO_Temp[1];
      AN    #Ctrl[0];
      AN    #Ctrl[1];
      AN    #McFlag;
      =     #DO_Temp[2];
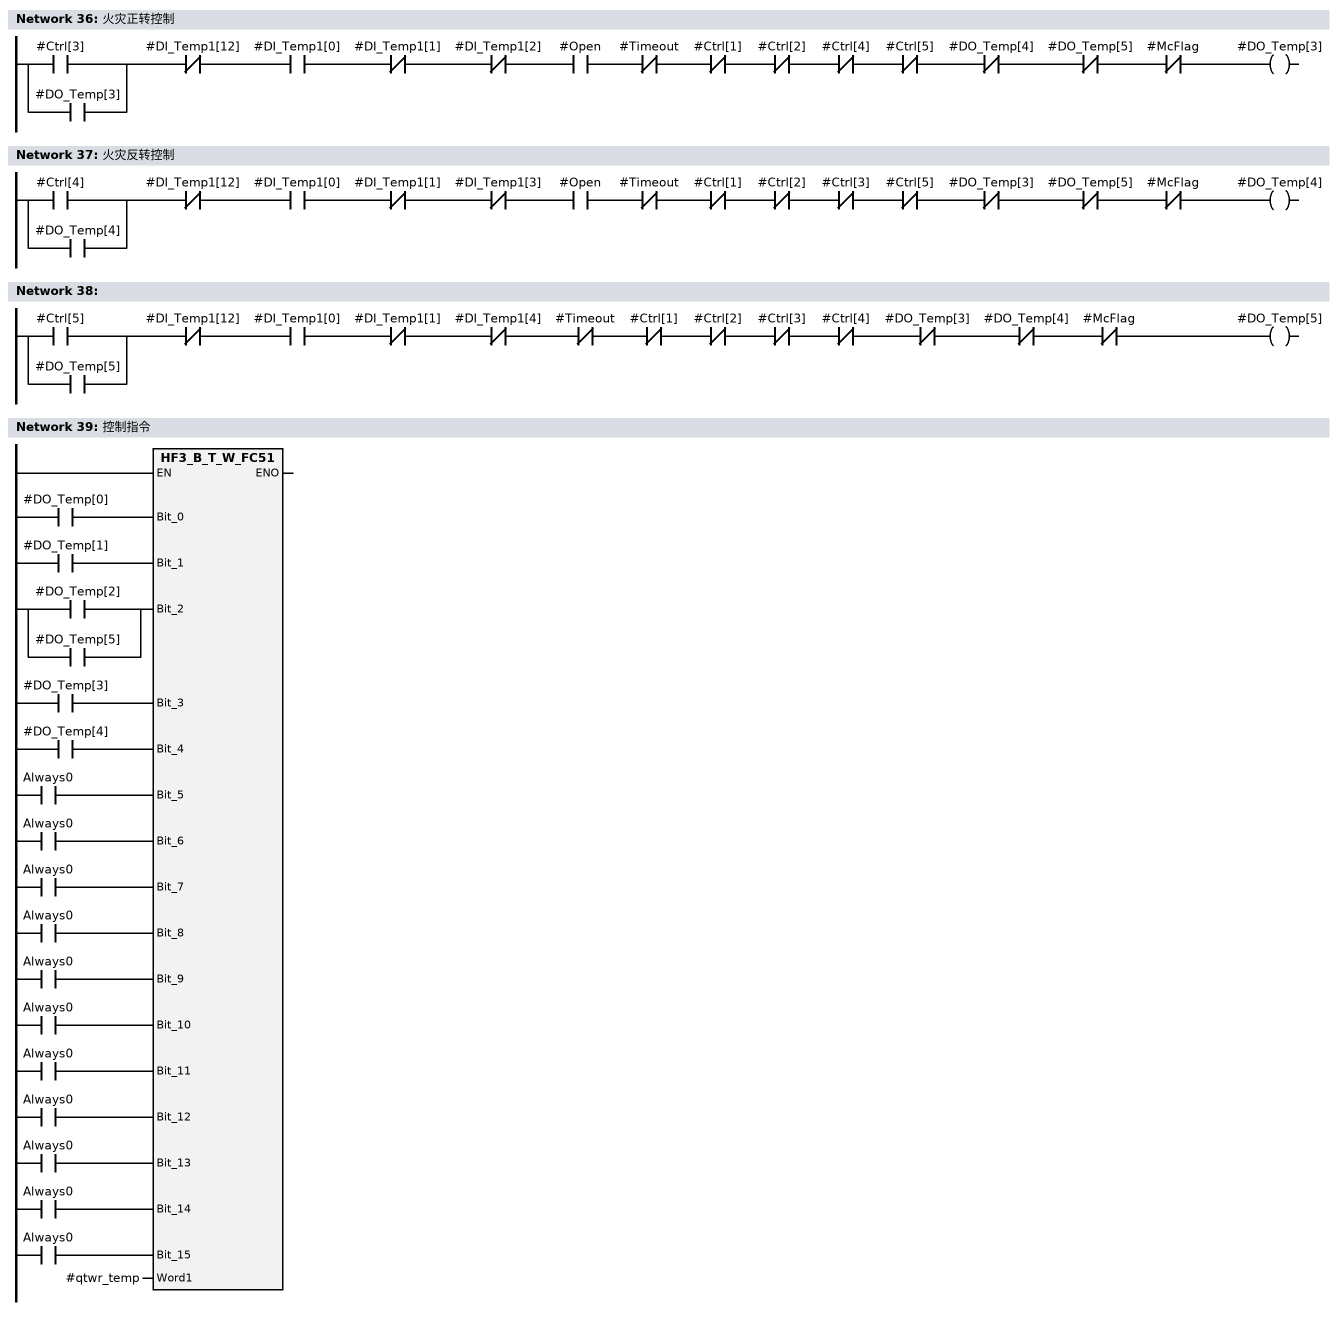
NETWORK
TITLE = 火灾正转控制
      A(;
      O     #Ctrl[3];
      O     #DO_Temp[3];
      );
      AN    #DI_Temp1[12];
      A     #DI_Temp1[0];
      AN    #DI_Temp1[1];
      AN    #DI_Temp1[2];
      A     #Open;
      AN    #Timeout;
      AN    #Ctrl[1];
      AN    #Ctrl[2];
      AN    #Ctrl[4];
      AN    #Ctrl[5];
      AN    #DO_Temp[4];
      AN    #DO_Temp[5];
      AN    #McFlag;
      =     #DO_Temp[3];
NETWORK
TITLE = 火灾反转控制
      A(;
      O     #Ctrl[4];
      O     #DO_Temp[4];
      );
      AN    #DI_Temp1[12];
      A     #DI_Temp1[0];
      AN    #DI_Temp1[1];
      AN    #DI_Temp1[3];
      A     #Open;
      AN    #Timeout;
      AN    #Ctrl[1];
      AN    #Ctrl[2];
      AN    #Ctrl[3];
      AN    #Ctrl[5];
      AN    #DO_Temp[3];
      AN    #DO_Temp[5];
      AN    #McFlag;
      =     #DO_Temp[4];
NETWORK
TITLE =
      A(;
      O     #Ctrl[5];
      O     #DO_Temp[5];
      );
      AN    #DI_Temp1[12];
      A     #DI_Temp1[0];
      AN    #DI_Temp1[1];
      AN    #DI_Temp1[4];
      AN    #Timeout;
      AN    #Ctrl[1];
      AN    #Ctrl[2];
      AN    #Ctrl[3];
      AN    #Ctrl[4];
      AN    #DO_Temp[3];
      AN    #DO_Temp[4];
      AN    #McFlag;
      =     #DO_Temp[5];
NETWORK
TITLE = 控制指令
      A     #DO_Temp[0];
      =     L 10.0;
      BLD   103;
      A     #DO_Temp[1];
      =     L 10.1;
      BLD   103;
      A(;
      O     #DO_Temp[2];
      O     #DO_Temp[5];
      );
      =     L 10.2;
      BLD   103;
      A     #DO_Temp[3];
      =     L 10.3;
      BLD   103;
      A     #DO_Temp[4];
      =     L 10.4;
      BLD   103;
      A     "Always0";
      =     L 10.5;
      BLD   103;
      A     "Always0";
      =     L 10.6;
      BLD   103;
      A     "Always0";
      =     L 10.7;
      BLD   103;
      A     "Always0";
      =     L 11.0;
      BLD   103;
      A     "Always0";
      =     L 11.1;
      BLD   103;
      A     "Always0";
      =     L 11.2;
      BLD   103;
      A     "Always0";
      =     L 11.3;
      BLD   103;
      A     "Always0";
      =     L 11.4;
      BLD   103;
      A     "Always0";
      =     L 11.5;
      BLD   103;
      A     "Always0";
      =     L 11.6;
      BLD   103;
      A     "Always0";
      =     L 11.7;
      BLD   103;
      CALL  "HF3_B_T_W_FC51" (
           Bit_0                    := L 10.0,
           Bit_1                    := L 10.1,
           Bit_2                    := L 10.2,
           Bit_3                    := L 10.3,
           Bit_4                    := L 10.4,
           Bit_5                    := L 10.5,
           Bit_6                    := L 10.6,
           Bit_7                    := L 10.7,
           Bit_8                    := L 11.0,
           Bit_9                    := L 11.1,
           Bit_10                   := L 11.2,
           Bit_11                   := L 11.3,
           Bit_12                   := L 11.4,
           Bit_13                   := L 11.5,
           Bit_14                   := L 11.6,
           Bit_15                   := L 11.7,
           Word1                    := #qtwr_temp);
      NOP   0;
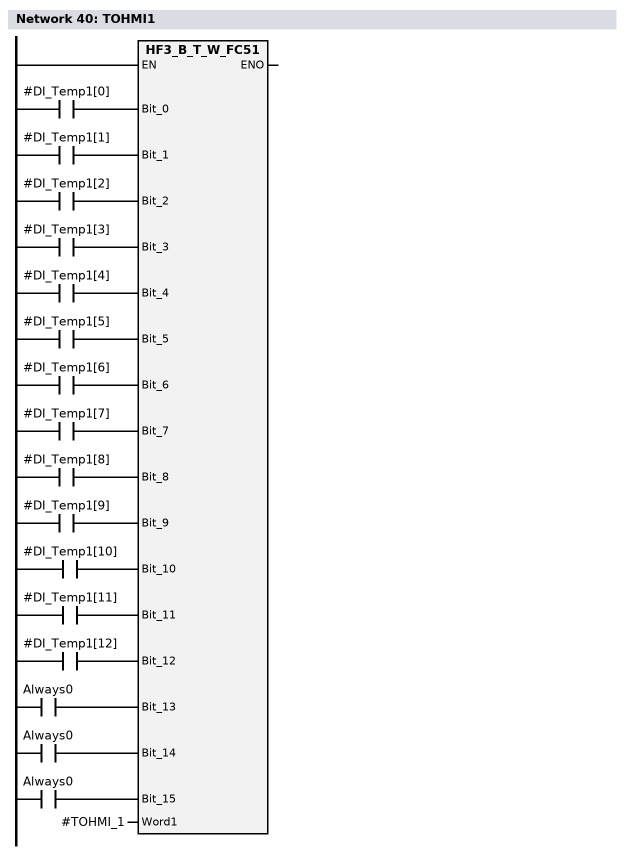
NETWORK
TITLE = TOHMI1
      A     #DI_Temp1[0];
      =     L 10.0;
      BLD   103;
      A     #DI_Temp1[1];
      =     L 10.1;
      BLD   103;
      A     #DI_Temp1[2];
      =     L 10.2;
      BLD   103;
      A     #DI_Temp1[3];
      =     L 10.3;
      BLD   103;
      A     #DI_Temp1[4];
      =     L 10.4;
      BLD   103;
      A     #DI_Temp1[5];
      =     L 10.5;
      BLD   103;
      A     #DI_Temp1[6];
      =     L 10.6;
      BLD   103;
      A     #DI_Temp1[7];
      =     L 10.7;
      BLD   103;
      A     #DI_Temp1[8];
      =     L 11.0;
      BLD   103;
      A     #DI_Temp1[9];
      =     L 11.1;
      BLD   103;
      A     #DI_Temp1[10];
      =     L 11.2;
      BLD   103;
      A     #DI_Temp1[11];
      =     L 11.3;
      BLD   103;
      A     #DI_Temp1[12];
      =     L 11.4;
      BLD   103;
      A     "Always0";
      =     L 11.5;
      BLD   103;
      A     "Always0";
      =     L 11.6;
      BLD   103;
      A     "Always0";
      =     L 11.7;
      BLD   103;
      CALL  "HF3_B_T_W_FC51" (
           Bit_0                    := L 10.0,
           Bit_1                    := L 10.1,
           Bit_2                    := L 10.2,
           Bit_3                    := L 10.3,
           Bit_4                    := L 10.4,
           Bit_5                    := L 10.5,
           Bit_6                    := L 10.6,
           Bit_7                    := L 10.7,
           Bit_8                    := L 11.0,
           Bit_9                    := L 11.1,
           Bit_10                   := L 11.2,
           Bit_11                   := L 11.3,
           Bit_12                   := L 11.4,
           Bit_13                   := L 11.5,
           Bit_14                   := L 11.6,
           Bit_15                   := L 11.7,
           Word1                    := #TOHMI_1);
      NOP   0;
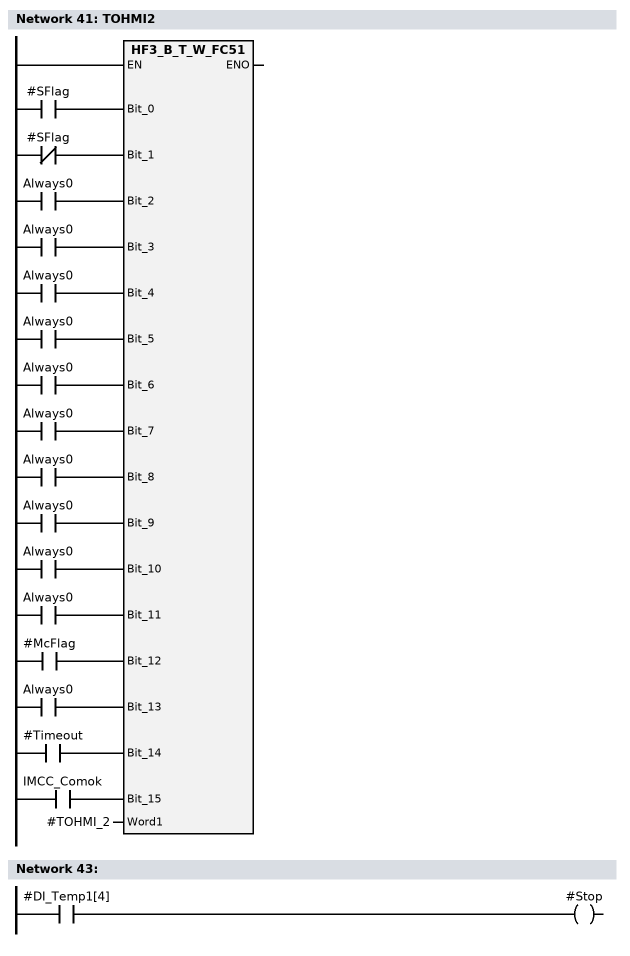
NETWORK
TITLE = TOHMI2
      A     #SFlag;
      =     L 10.0;
      BLD   103;
      AN    #SFlag;
      =     L 10.1;
      BLD   103;
      A     "Always0";
      =     L 10.2;
      BLD   103;
      A     "Always0";
      =     L 10.3;
      BLD   103;
      A     "Always0";
      =     L 10.4;
      BLD   103;
      A     "Always0";
      =     L 10.5;
      BLD   103;
      A     "Always0";
      =     L 10.6;
      BLD   103;
      A     "Always0";
      =     L 10.7;
      BLD   103;
      A     "Always0";
      =     L 11.0;
      BLD   103;
      A     "Always0";
      =     L 11.1;
      BLD   103;
      A     "Always0";
      =     L 11.2;
      BLD   103;
      A     "Always0";
      =     L 11.3;
      BLD   103;
      A     #McFlag;
      =     L 11.4;
      BLD   103;
      A     "Always0";
      =     L 11.5;
      BLD   103;
      A     #Timeout;
      =     L 11.6;
      BLD   103;
      A     "IMCC_Comok";
      =     L 11.7;
      BLD   103;
      CALL  "HF3_B_T_W_FC51" (
           Bit_0                    := L 10.0,
           Bit_1                    := L 10.1,
           Bit_2                    := L 10.2,
           Bit_3                    := L 10.3,
           Bit_4                    := L 10.4,
           Bit_5                    := L 10.5,
           Bit_6                    := L 10.6,
           Bit_7                    := L 10.7,
           Bit_8                    := L 11.0,
           Bit_9                    := L 11.1,
           Bit_10                   := L 11.2,
           Bit_11                   := L 11.3,
           Bit_12                   := L 11.4,
           Bit_13                   := L 11.5,
           Bit_14                   := L 11.6,
           Bit_15                   := L 11.7,
           Word1                    := #TOHMI_2);
      NOP   0;
NETWORK
TITLE = 信号输出
//控制命令输出
      CLR;
      L     #SCtrl;
      L     W#16#ABCD;
      <>I;
      JC    seiz;
      L     W#16#0;
      T     #qtwr_temp;
seiz: L     #qtwr_temp;
      T     #qtWR;
//tohmi输出
      L     #HMI_Adr;
      SLD   3;
      LAR1;
      OPN   DB [#DB_NO];
      L     #TOHMI_1;
      T     DBW [AR1,P#0.0];
      L     #TOHMI_2;
      T     DBW [AR1,P#2.0];
NETWORK
TITLE =
      A     #DI_Temp1[4];
      =     #Stop;
NETWORK
TITLE =
      A(;
      O     #DI_Temp1[2];
      O     #DI_Temp1[3];
      );
      =     L 10.0;
      BLD   103;
      A     #Flt;
      =     L 10.1;
      BLD   103;
      A     M 20.3;
      =     L 10.2;
      BLD   103;
      A     #SCtrl_Temp[12];
      =     L 10.4;
      BLD   103;
      A     #SCtrl_Temp[13];
      =     L 10.5;
      BLD   103;
      BLD   14;
      =     L 17.0;
      L     DINO;
      T     LW 15;
      CDB;
      OPN   DI [LW 15];
      TAR2  LD 11;
      A     L 10.0;
      =     DIX [AR2,P#176.0];
      A     L 10.1;
      =     DIX [AR2,P#176.1];
      A     L 10.2;
      =     DIX [AR2,P#176.2];
      A     L 10.4;
      =     DIX [AR2,P#176.4];
      A     L 10.5;
      =     DIX [AR2,P#176.5];
      +AR2  P#176.0;
      UC    "HF3_RunFaultSum";
      LAR2  LD 11;
      L     DID [AR2,P#178.0];
      T     DBD [AR2,P#52.0];
      L     DIW [AR2,P#182.0];
      T     DBW [AR2,P#58.0];
      L     DIW [AR2,P#184.0];
      T     DBW [AR2,P#56.0];
      CDB;
      BLD   15;
      NOP   0;
END_FUNCTION_BLOCK

FUNCTION_BLOCK "HF3_IMCC_TEF_FB2661"	// FB 2661
VERSION : 0.1
VAR
  PT : TIME  := T#45S;
  UOF_A1 : FB 2662;
END_VAR
BEGIN
NETWORK
TITLE =
// (network holds code this reader does not know; not shown)
END_FUNCTION_BLOCK

FUNCTION_BLOCK "HF3_IMCC_TEF_FB2662"	// FB 2662
VERSION : 0.1
VAR_INPUT
  Main : BOOL ;	//1为大端  0为小端
  IN_RD : ARRAY  [0 .. 14 ] OF WORD ;
  HMI_Adr : INT ;
  SCtrl : WORD ;	//0单控 1模控 2启动 3停止 6火灾
  MCtrl : ARRAY  [0 .. 3 ] OF //模式控制
  BOOL ;
  Mode : ARRAY  [0 .. 15 ] OF //模式执行状态
  BOOL ;
  Open : BOOL ;	//风阀开连锁
  PT : TIME ;	//执行时间
  ALL : ARRAY  [0 .. 15 ] OF //单系统命令
  BOOL ;
  H_P_All_Ctrl : WORD ;	//全局命令
  FireAlarm : BOOL ;	//火灾报警
  BlockAlarm : BOOL ;	//阻塞报警
  ManuSet : INT ;	//手动频率给定
END_VAR
VAR_OUTPUT
  qnWR : ARRAY  [0 .. 1 ] OF WORD ;
  RT : REAL ;	//运行时间
  SumFlt : INT ;	//故障次数
  SumRun : INT ;	//启动次数
  Refuse : BOOL ;	//模式不符
  Stop : BOOL ;	//风机控制
END_VAR
VAR
  IN_RD1 : WORD ;
  qtWR : WORD ;
  TOHMI_1 : WORD ;
  TOHMI_2 : WORD ;
  qtwr_temp : WORD ;
  SFlag : BOOL ;	//单控标志
  McFlag : BOOL ;	//检修牌
  QTout : BOOL ;	//输出超时
  SingTout : BOOL ;	//单控超时
  Timeout : BOOL ;	//设备动作超时
  Flt : BOOL ;	//设备综合故障
  PID_EN : BOOL ;	//pid使能
  Fault : BOOL ;	//故障
  sCFRun : BOOL ;
  sCFStop : BOOL ;
  INPUT1 : ARRAY  [0 .. 15 ] OF //设备状态字
  BOOL ;
  OUTPUT : ARRAY  [0 .. 15 ] OF //输出状态字
  BOOL ;
  Ctrl : ARRAY  [0 .. 15 ] OF BOOL ;
  SCtrl_Temp : ARRAY  [0 .. 15 ] OF //HMI命令
  BOOL ;
  Latch : ARRAY  [0 .. 7 ] OF BOOL ;
  h_P_all_temp : ARRAY  [0 .. 15 ] OF BOOL ;
  ton1 : SFB 4;
  ton2 : SFB 4;
  RunFaultSum : FB 2006;
  PID_TEF : FB 2005;
END_VAR
VAR_TEMP
  AR2_Value : DWORD ;
  DI_NO : INT ;
  Data_Len : INT ;
  DB_NO : INT ;
END_VAR
BEGIN
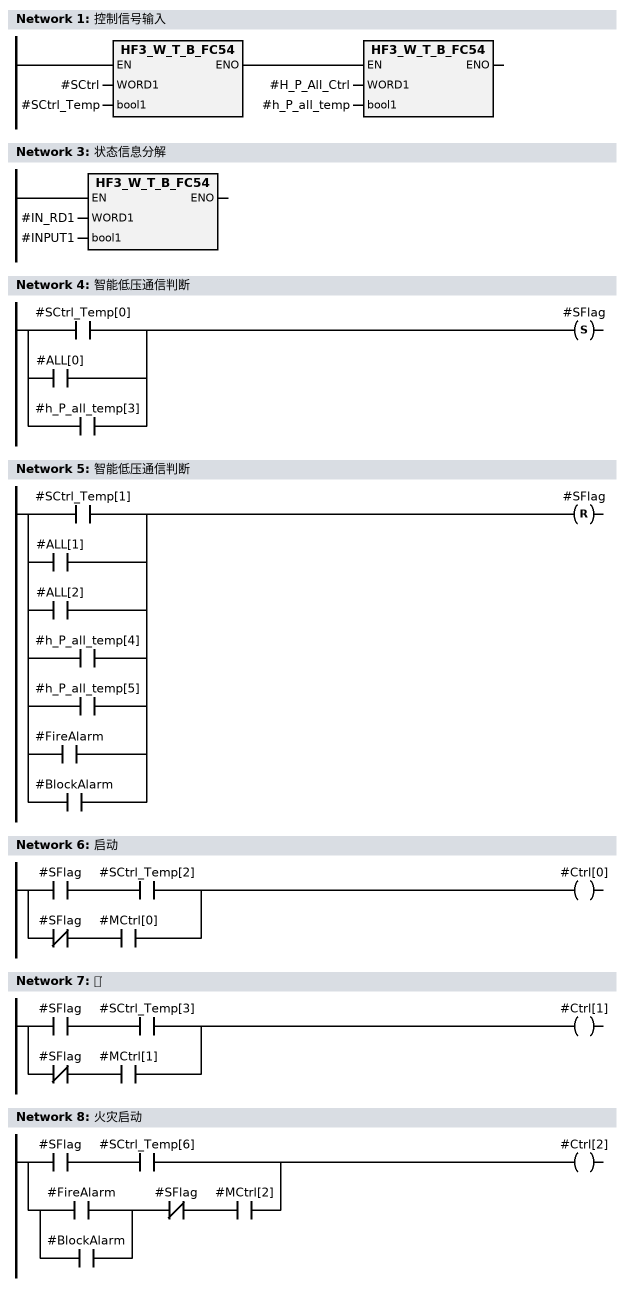
NETWORK
TITLE = 控制信号输入
      A(;
      CALL  "HF3_W_T_B_FC54" (
           WORD1                    := #SCtrl,
           bool1                    := #SCtrl_Temp);
      A     BR;
      );
      JNB   _001;
      CALL  "HF3_W_T_B_FC54" (
           WORD1                    := #H_P_All_Ctrl,
           bool1                    := #h_P_all_temp);
_001: NOP   0;
NETWORK
TITLE = 状态信息读取
//
//第1个字BIT 0BAS
//第1个字BIT 1就地
//第1个字BIT 2变频/工频开关位置
//第1个字BIT 3变频运行状态
//第1个字BIT 4工频运行状态
//第1个字BIT 5停止状态
//第1个字BIT 6变频器故障
//第1个字BIT 7振动超高报警
//第1个字BIT 8轴承温度报警
//第1个字BIT 9绕组温度报警
//第1个字BIT 10变频器过载
//第1个字BIT 11电动机缺相
//第1个字BIT 12火灾切除保护
//
//
//第2个字频率反馈
//第3个字电动机电流A
//第4个字电动机电流B
//第5个字电动机电流C
//第6个字电动机电压A
//第7个字电动机电压B
//第8个字电动机电压C
//第9个字前轴承温度
//第10个字后轴承温度
//第11个字绕组温度A
//第12个字绕组温度B
//第13个字绕组温度C
//第14个字水平振动
//第15个字垂直振动
//
      TAR2;
      T     #AR2_Value;
      L     6002;
      T     #DB_NO;
      A     #Main;	//此端是否为大端
      JC    big;
      L     6004;
      T     #DB_NO;
big:  L     DINO;	//存储背景数据块号
      T     #DI_NO;
      OPN   DB [#DB_NO];	//打开
      L     #HMI_Adr;
      SLD   3;
      LAR1;
// *********************排热风机中DI状态读取**********************
      L     #IN_RD[0];	//第一个字中包含数字量信息
      T     #IN_RD1;
//初始化AR2寄存器用于AI量传递
      TAR2;
      AD    DW#16#FFFFFF;
      L     P##IN_RD;
      +D;
      OD    DW#16#85000000;
      LAR2;
//*********************排热风机中AI状态读取**********************
//读取模拟量输入
      L     14;
ilop: T     #Data_Len;
      L     W [AR2,P#2.0];	//智能低压点表新更新，第二个字开始为模拟量
      T     DBW [AR1,P#4.0];
      +AR1  P#2.0;
      +AR2  P#2.0;
      L     #Data_Len;
      LOOP  ilop;
//恢复AR2 DI寄存器
      L     #AR2_Value;
      LAR2;
//     OPN   DI [#DI_NO]
NETWORK
TITLE = 状态信息分解
      CALL  "HF3_W_T_B_FC54" (
           WORD1                    := #IN_RD1,
           bool1                    := #INPUT1);
      NOP   0;
NETWORK
TITLE = 智能低压通信判断
      O     #SCtrl_Temp[0];
      O     #ALL[0];
      O     #h_P_all_temp[3];
      S     #SFlag;
NETWORK
TITLE = 智能低压通信判断
      O     #SCtrl_Temp[1];
      O     #ALL[1];
      O     #ALL[2];
      O     #h_P_all_temp[4];
      O     #h_P_all_temp[5];
      O     #FireAlarm;
      O     #BlockAlarm;
      R     #SFlag;
NETWORK
TITLE = 启动
      A     #SFlag;
      A     #SCtrl_Temp[2];
      O;
      AN    #SFlag;
      A     #MCtrl[0];
      =     #Ctrl[0];
NETWORK
TITLE = ֹͣ
      A     #SFlag;
      A     #SCtrl_Temp[3];
      O;
      AN    #SFlag;
      A     #MCtrl[1];
      =     #Ctrl[1];
NETWORK
TITLE = 火灾启动
      A     #SFlag;
      A     #SCtrl_Temp[6];
      O;
      A(;
      O     #FireAlarm;
      O     #BlockAlarm;
      );
      AN    #SFlag;
      A     #MCtrl[2];
      =     #Ctrl[2];
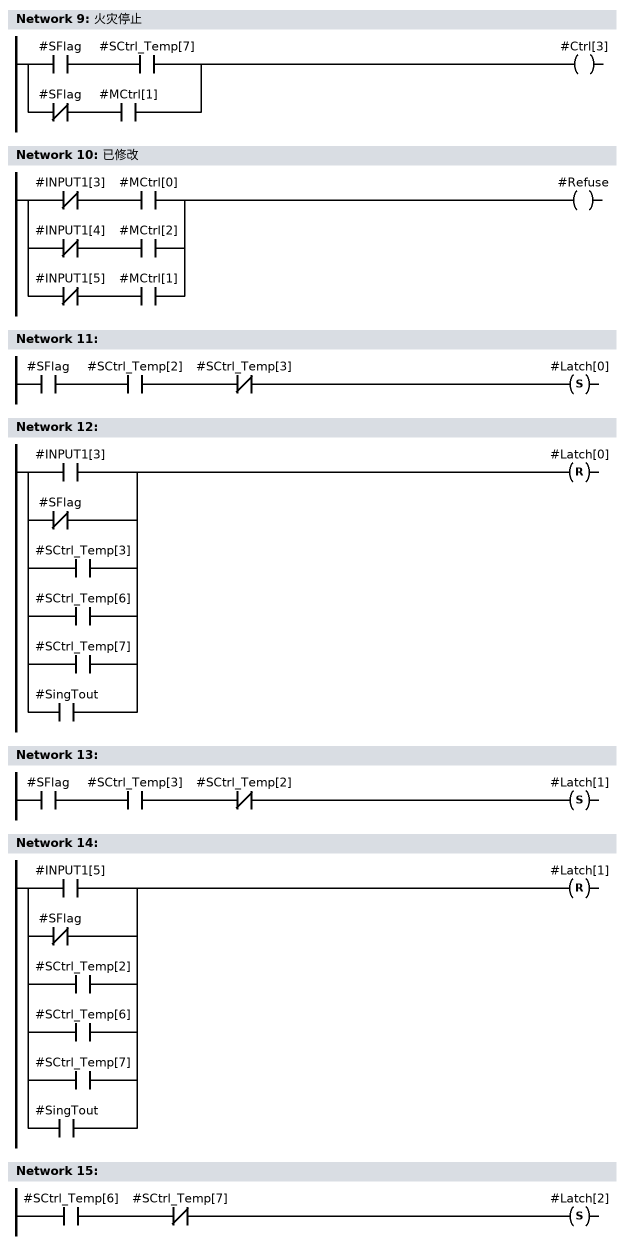
NETWORK
TITLE = 火灾停止
      A     #SFlag;
      A     #SCtrl_Temp[7];
      O;
      AN    #SFlag;
      A     #MCtrl[1];
      =     #Ctrl[3];
NETWORK
TITLE = 已修改
      AN    #INPUT1[3];
      A     #MCtrl[0];
      O;
      AN    #INPUT1[4];
      A     #MCtrl[2];
      O;
      AN    #INPUT1[5];
      A     #MCtrl[1];
      =     #Refuse;
NETWORK
TITLE =
      A     #SFlag;
      A     #SCtrl_Temp[2];
      AN    #SCtrl_Temp[3];
      S     #Latch[0];
NETWORK
TITLE =
      O     #INPUT1[3];
      ON    #SFlag;
      O     #SCtrl_Temp[3];
      O     #SCtrl_Temp[6];
      O     #SCtrl_Temp[7];
      O     #SingTout;
      R     #Latch[0];
NETWORK
TITLE =
      A     #SFlag;
      A     #SCtrl_Temp[3];
      AN    #SCtrl_Temp[2];
      S     #Latch[1];
NETWORK
TITLE =
      O     #INPUT1[5];
      ON    #SFlag;
      O     #SCtrl_Temp[2];
      O     #SCtrl_Temp[6];
      O     #SCtrl_Temp[7];
      O     #SingTout;
      R     #Latch[1];
NETWORK
TITLE =
      A     #SCtrl_Temp[6];
      AN    #SCtrl_Temp[7];
      S     #Latch[2];
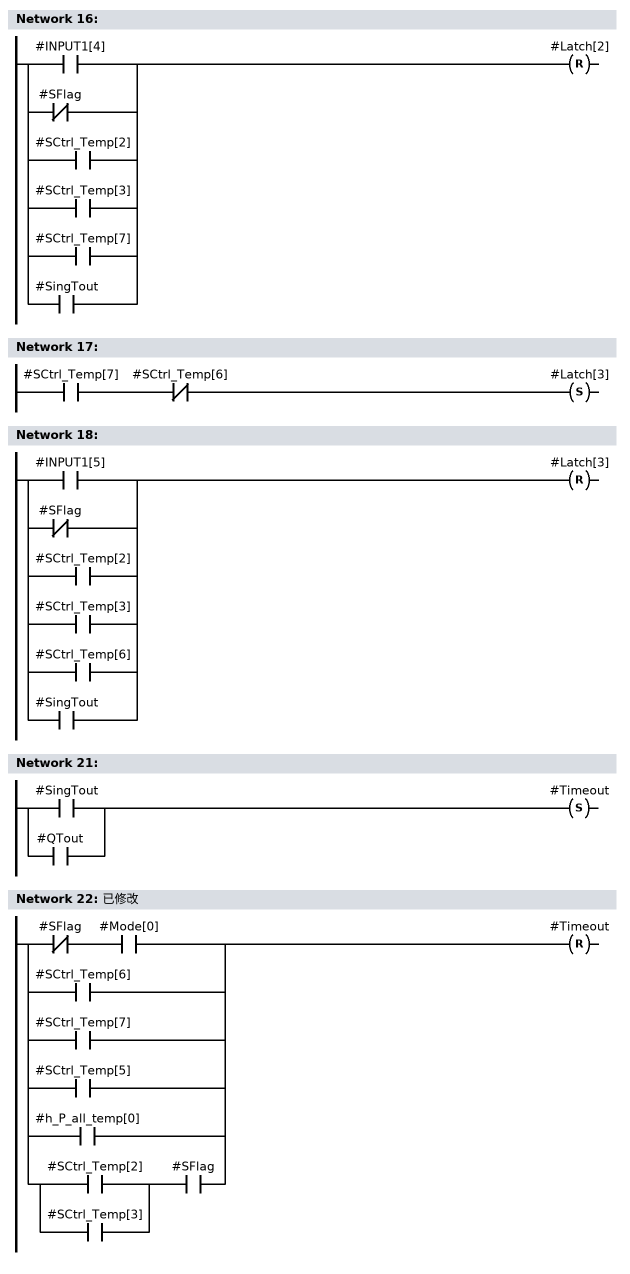
NETWORK
TITLE =
      O     #INPUT1[4];
      ON    #SFlag;
      O     #SCtrl_Temp[2];
      O     #SCtrl_Temp[3];
      O     #SCtrl_Temp[7];
      O     #SingTout;
      R     #Latch[2];
NETWORK
TITLE =
      A     #SCtrl_Temp[7];
      AN    #SCtrl_Temp[6];
      S     #Latch[3];
NETWORK
TITLE =
      O     #INPUT1[5];
      ON    #SFlag;
      O     #SCtrl_Temp[2];
      O     #SCtrl_Temp[3];
      O     #SCtrl_Temp[6];
      O     #SingTout;
      R     #Latch[3];
NETWORK
TITLE =
      A(;
      O     #Latch[0];
      O     #Latch[1];
      O     #Latch[2];
      O     #Latch[3];
      );
      =     L 10.0;
      BLD   103;
      BLD   16;
      =     L 17.0;
      L     DINO;
      T     LW 15;
      CDB;
      OPN   DI [LW 15];
      TAR2  LD 11;
      A     L 10.0;
      =     DIX [AR2,P#92.0];
      L     DBD [AR2,P#42.0];
      T     DID [AR2,P#94.0];
      +AR2  P#92.0;
      UC    "TON";
      LAR2  LD 11;
      A     DIX [AR2,P#98.0];
      =     DBX [AR2,P#78.3];
      CDB;
      BLD   17;
      NOP   0;
NETWORK
TITLE =
      A(;
      O     #OUTPUT[0];
      O     #OUTPUT[1];
      O     #sCFRun;
      O     #sCFStop;
      );
      =     L 10.0;
      BLD   103;
      BLD   16;
      =     L 17.0;
      L     DINO;
      T     LW 15;
      CDB;
      OPN   DI [LW 15];
      TAR2  LD 11;
      A     L 10.0;
      =     DIX [AR2,P#114.0];
      L     DBD [AR2,P#42.0];
      T     DID [AR2,P#116.0];
      +AR2  P#114.0;
      UC    "TON";
      LAR2  LD 11;
      A     DIX [AR2,P#120.0];
      =     DBX [AR2,P#78.2];
      CDB;
      BLD   17;
      NOP   0;
NETWORK
TITLE =
      O     #SingTout;
      O     #QTout;
      S     #Timeout;
NETWORK
TITLE = 已修改
      AN    #SFlag;
      A     #Mode[0];
      O     #SCtrl_Temp[6];
      O     #SCtrl_Temp[7];
      O     #SCtrl_Temp[5];
      O     #h_P_all_temp[0];
      O;
      A(;
      O     #SCtrl_Temp[2];
      O     #SCtrl_Temp[3];
      );
      A     #SFlag;
      R     #Timeout;
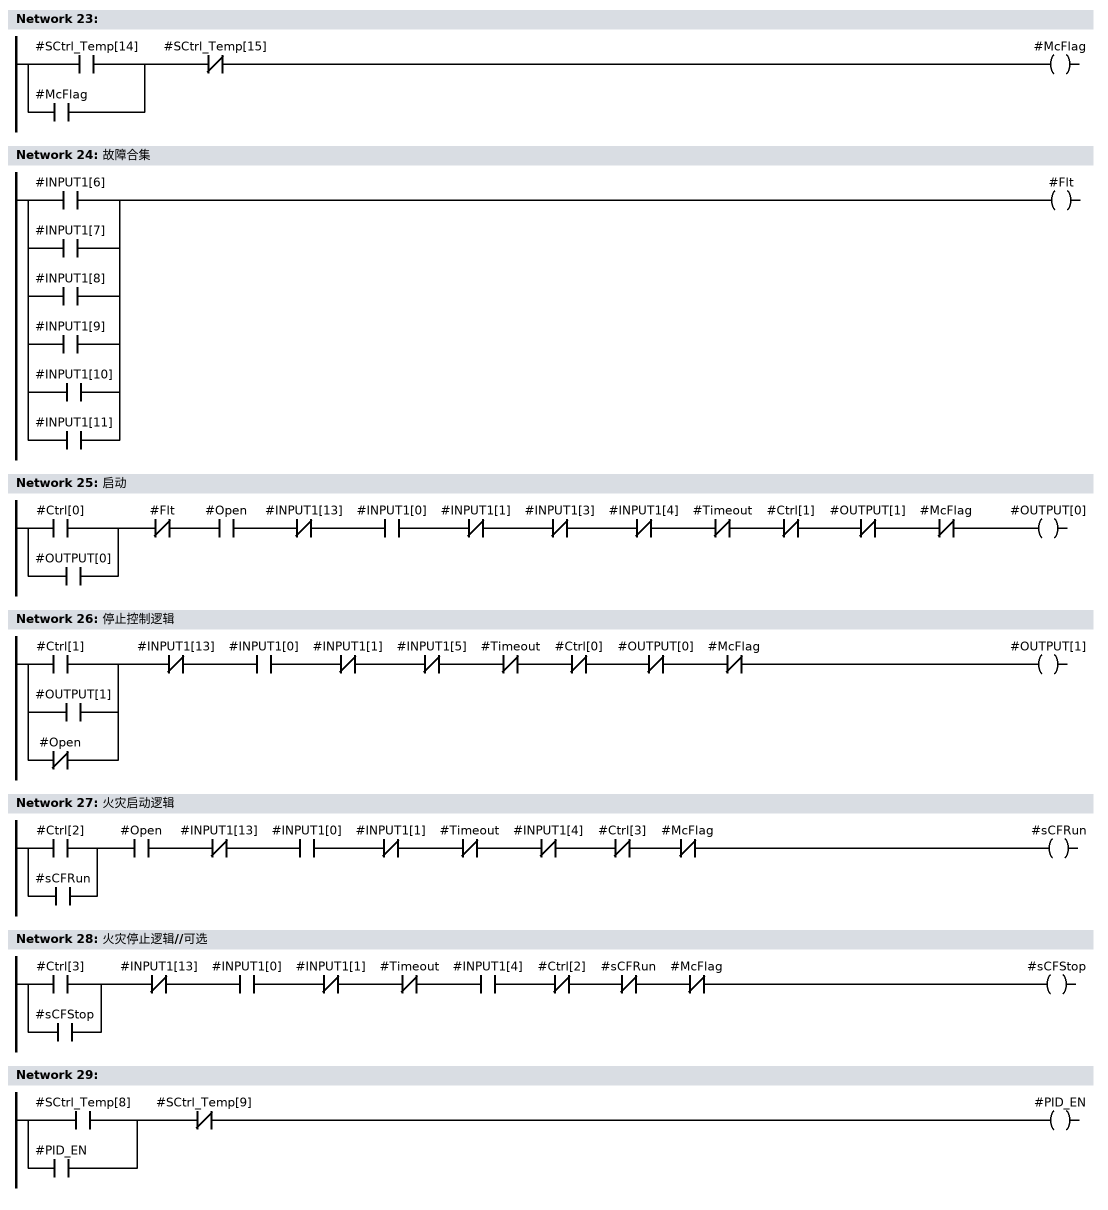
NETWORK
TITLE =
      A(;
      O     #SCtrl_Temp[14];
      O     #McFlag;
      );
      AN    #SCtrl_Temp[15];
      =     #McFlag;
NETWORK
TITLE = 故障合集
      O     #INPUT1[6];
      O     #INPUT1[7];
      O     #INPUT1[8];
      O     #INPUT1[9];
      O     #INPUT1[10];
      O     #INPUT1[11];
      =     #Flt;
NETWORK
TITLE = 启动
      A(;
      O     #Ctrl[0];
      O     #OUTPUT[0];
      );
      AN    #Flt;
      A     #Open;
      AN    #INPUT1[13];
      A     #INPUT1[0];
      AN    #INPUT1[1];
      AN    #INPUT1[3];
      AN    #INPUT1[4];
      AN    #Timeout;
      AN    #Ctrl[1];
      AN    #OUTPUT[1];
      AN    #McFlag;
      =     #OUTPUT[0];
NETWORK
TITLE = 停止控制逻辑
      A(;
      O     #Ctrl[1];
      O     #OUTPUT[1];
      ON    #Open;
      );
      AN    #INPUT1[13];
      A     #INPUT1[0];
      AN    #INPUT1[1];
      AN    #INPUT1[5];
      AN    #Timeout;
      AN    #Ctrl[0];
      AN    #OUTPUT[0];
      AN    #McFlag;
      =     #OUTPUT[1];
NETWORK
TITLE = 火灾启动逻辑
      A(;
      O     #Ctrl[2];
      O     #sCFRun;
      );
      A     #Open;
      AN    #INPUT1[13];
      A     #INPUT1[0];
      AN    #INPUT1[1];
      AN    #Timeout;
      AN    #INPUT1[4];
      AN    #Ctrl[3];
      AN    #McFlag;
      =     #sCFRun;
NETWORK
TITLE = 火灾停止逻辑//可选
      A(;
      O     #Ctrl[3];
      O     #sCFStop;
      );
      AN    #INPUT1[13];
      A     #INPUT1[0];
      AN    #INPUT1[1];
      AN    #Timeout;
      A     #INPUT1[4];
      AN    #Ctrl[2];
      AN    #sCFRun;
      AN    #McFlag;
      =     #sCFStop;
NETWORK
TITLE =
      A(;
      O     #SCtrl_Temp[8];
      O     #PID_EN;
      );
      AN    #SCtrl_Temp[9];
      =     #PID_EN;
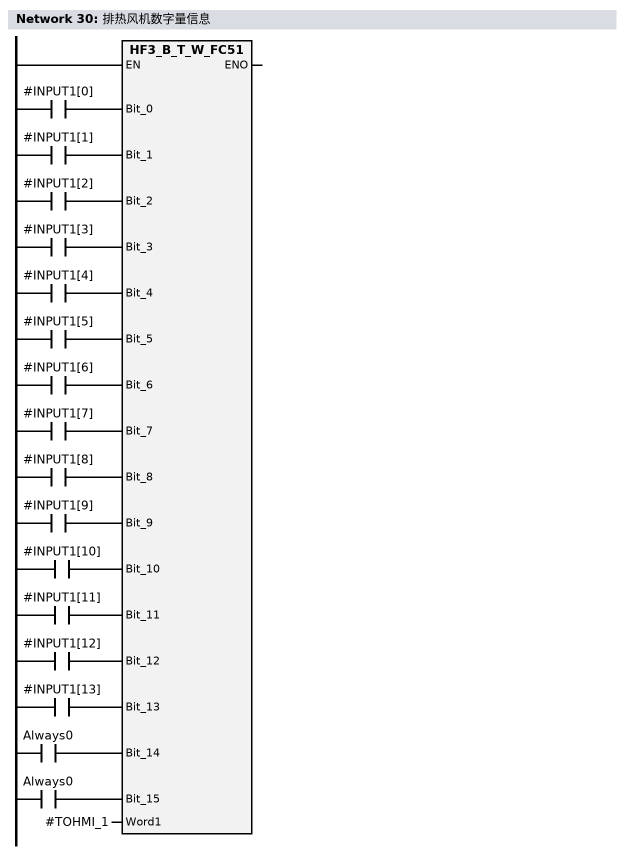
NETWORK
TITLE = 排热风机数字量信息
      A     #INPUT1[0];
      =     L 10.0;
      BLD   103;
      A     #INPUT1[1];
      =     L 10.1;
      BLD   103;
      A     #INPUT1[2];
      =     L 10.2;
      BLD   103;
      A     #INPUT1[3];
      =     L 10.3;
      BLD   103;
      A     #INPUT1[4];
      =     L 10.4;
      BLD   103;
      A     #INPUT1[5];
      =     L 10.5;
      BLD   103;
      A     #INPUT1[6];
      =     L 10.6;
      BLD   103;
      A     #INPUT1[7];
      =     L 10.7;
      BLD   103;
      A     #INPUT1[8];
      =     L 11.0;
      BLD   103;
      A     #INPUT1[9];
      =     L 11.1;
      BLD   103;
      A     #INPUT1[10];
      =     L 11.2;
      BLD   103;
      A     #INPUT1[11];
      =     L 11.3;
      BLD   103;
      A     #INPUT1[12];
      =     L 11.4;
      BLD   103;
      A     #INPUT1[13];
      =     L 11.5;
      BLD   103;
      A     "Always0";
      =     L 11.6;
      BLD   103;
      A     "Always0";
      =     L 11.7;
      BLD   103;
      CALL  "HF3_B_T_W_FC51" (
           Bit_0                    := L 10.0,
           Bit_1                    := L 10.1,
           Bit_2                    := L 10.2,
           Bit_3                    := L 10.3,
           Bit_4                    := L 10.4,
           Bit_5                    := L 10.5,
           Bit_6                    := L 10.6,
           Bit_7                    := L 10.7,
           Bit_8                    := L 11.0,
           Bit_9                    := L 11.1,
           Bit_10                   := L 11.2,
           Bit_11                   := L 11.3,
           Bit_12                   := L 11.4,
           Bit_13                   := L 11.5,
           Bit_14                   := L 11.6,
           Bit_15                   := L 11.7,
           Word1                    := #TOHMI_1);
      NOP   0;
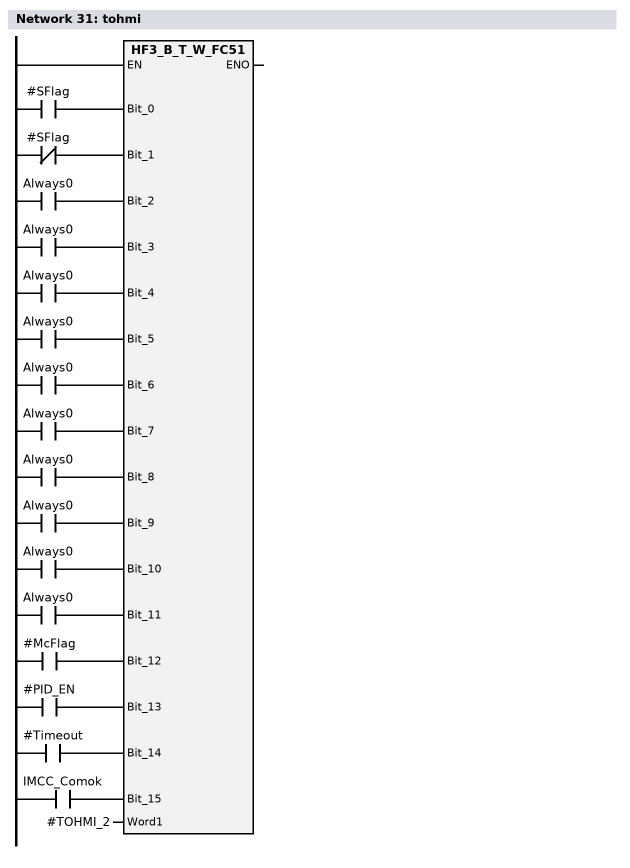
NETWORK
TITLE = tohmi
      A     #SFlag;
      =     L 10.0;
      BLD   103;
      AN    #SFlag;
      =     L 10.1;
      BLD   103;
      A     "Always0";
      =     L 10.2;
      BLD   103;
      A     "Always0";
      =     L 10.3;
      BLD   103;
      A     "Always0";
      =     L 10.4;
      BLD   103;
      A     "Always0";
      =     L 10.5;
      BLD   103;
      A     "Always0";
      =     L 10.6;
      BLD   103;
      A     "Always0";
      =     L 10.7;
      BLD   103;
      A     "Always0";
      =     L 11.0;
      BLD   103;
      A     "Always0";
      =     L 11.1;
      BLD   103;
      A     "Always0";
      =     L 11.2;
      BLD   103;
      A     "Always0";
      =     L 11.3;
      BLD   103;
      A     #McFlag;
      =     L 11.4;
      BLD   103;
      A     #PID_EN;
      =     L 11.5;
      BLD   103;
      A     #Timeout;
      =     L 11.6;
      BLD   103;
      A     "IMCC_Comok";
      =     L 11.7;
      BLD   103;
      CALL  "HF3_B_T_W_FC51" (
           Bit_0                    := L 10.0,
           Bit_1                    := L 10.1,
           Bit_2                    := L 10.2,
           Bit_3                    := L 10.3,
           Bit_4                    := L 10.4,
           Bit_5                    := L 10.5,
           Bit_6                    := L 10.6,
           Bit_7                    := L 10.7,
           Bit_8                    := L 11.0,
           Bit_9                    := L 11.1,
           Bit_10                   := L 11.2,
           Bit_11                   := L 11.3,
           Bit_12                   := L 11.4,
           Bit_13                   := L 11.5,
           Bit_14                   := L 11.6,
           Bit_15                   := L 11.7,
           Word1                    := #TOHMI_2);
      NOP   0;
